  A_360_01_SQ4_A428_7_VOL : FbAnalogInput_Medium (2094) := (                _sDescription := 'Faktisk luftmengde',                 _rCov_Increment := 1,                 _eUnits := WagoTypesBacnet.eBACnetUnits.UNIT_CUBIC_METERS_PER_HOUR           );
  A_360_01_SQ4_A428_7_SP : FbAnalogValue_Medium (2141) := (                _sDescription := 'Settpunkt',                 _rCov_Increment := 1,                 _eUnits := WagoTypesBacnet.eBACnetUnits.UNIT_CUBIC_METERS_PER_HOUR           );
  A_360_01_SQ4_A428_7_VMIN : FbAnalogValue_Medium (2142) := (                _sDescription := 'Minste luftmengde',                 _rCov_Increment := 1,                 _eUnits := WagoTypesBacnet.eBACnetUnits.UNIT_CUBIC_METERS_PER_HOUR           );
  A_360_01_SQ4_A428_7_VMAX : FbAnalogValue_Medium (2143) := (                _sDescription := 'Største luftmengde',                 _rCov_Increment := 1,                 _eUnits := WagoTypesBacnet.eBACnetUnits.UNIT_CUBIC_METERS_PER_HOUR           );
  A_360_01_SQ4_A428_7_FB : FbAnalogInput_Medium (2095) := (                _sDescription := 'Spjeldvinkel',                 _rCov_Increment := 1,                 _eUnits := WagoTypesBacnet.eBACnetUnits.UNIT_PERCENT           );
  A_360_01_SQ4_A428_7_C : FbAnalogOutput_Medium (2047) := (                _sDescription := 'Pådrag',                 _rCov_Increment := 1,                 _eUnits := WagoTypesBacnet.eBACnetUnits.UNIT_PERCENT           );
  A_360_01_SQ4_A428_7_KMD : FbMultiStateValue_Large (2047) := (                _sDescription := 'Manuell overstyring',                 _udiNumberOfStates := 8           );
  A_360_01_SQ4_A428_7_OPT_EKSKL : FbBinaryValue_Medium (2047) := (                _sDescription := 'Optimizer',                 _sActiveText := 'Utkoblet',                 _sInactiveText := 'Innkoblet'           );
  A_360_01_SQ4_A428_7_A1 : FbBinaryInput_Large (2094) := (                _sDescription := 'Luftmengde Sjeld',                 _sActiveText := 'Feil på luftmengde',                 _sInactiveText := 'Ingen feil',                 _udiNotificationClass := 22           );
  A_360_01_SQ4_A428_7_A2 : FbBinaryInput_Large (2095) := (                _sDescription := 'Kommunikasjonovervåking',                 _sActiveText := 'Kommunikasjonsfeil',                 _sInactiveText := 'Ingen feil',                 _udiNotificationClass := 22           );
  B_360_02_SQ5_UBH1_VOL : FbAnalogInput_Medium (2096) := (                _sDescription := 'Faktisk luftmengde',                 _rCov_Increment := 1,                 _eUnits := WagoTypesBacnet.eBACnetUnits.UNIT_CUBIC_METERS_PER_HOUR           );
  B_360_02_SQ5_UBH1_SP : FbAnalogValue_Medium (2144) := (                _sDescription := 'Settpunkt',                 _rCov_Increment := 1,                 _eUnits := WagoTypesBacnet.eBACnetUnits.UNIT_CUBIC_METERS_PER_HOUR           );
  B_360_02_SQ5_UBH1_VMIN : FbAnalogValue_Medium (2145) := (                _sDescription := 'Minste luftmengde',                 _rCov_Increment := 1,                 _eUnits := WagoTypesBacnet.eBACnetUnits.UNIT_CUBIC_METERS_PER_HOUR           );
  B_360_02_SQ5_UBH1_VMAX : FbAnalogValue_Medium (2146) := (                _sDescription := 'Største luftmengde',                 _rCov_Increment := 1,                 _eUnits := WagoTypesBacnet.eBACnetUnits.UNIT_CUBIC_METERS_PER_HOUR           );
  B_360_02_SQ5_UBH1_FB : FbAnalogInput_Medium (2097) := (                _sDescription := 'Spjeldvinkel',                 _rCov_Increment := 1,                 _eUnits := WagoTypesBacnet.eBACnetUnits.UNIT_PERCENT           );
  B_360_02_SQ5_UBH1_C : FbAnalogOutput_Medium (2048) := (                _sDescription := 'Pådrag',                 _rCov_Increment := 1,                 _eUnits := WagoTypesBacnet.eBACnetUnits.UNIT_PERCENT           );
  B_360_02_SQ5_UBH1_KMD : FbMultiStateValue_Large (2048) := (                _sDescription := 'Manuell overstyring',                 _udiNumberOfStates := 8           );
  B_360_02_SQ5_UBH1_OPT_EKSKL : FbBinaryValue_Medium (2048) := (                _sDescription := 'Optimizer',                 _sActiveText := 'Utkoblet',                 _sInactiveText := 'Innkoblet'           );
  B_360_02_SQ5_UBH1_A1 : FbBinaryInput_Large (2096) := (                _sDescription := 'Luftmengde Sjeld',                 _sActiveText := 'Feil på luftmengde',                 _sInactiveText := 'Ingen feil',                 _udiNotificationClass := 22           );
  B_360_02_SQ5_UBH1_A2 : FbBinaryInput_Large (2097) := (                _sDescription := 'Kommunikasjonovervåking',                 _sActiveText := 'Kommunikasjonsfeil',                 _sInactiveText := 'Ingen feil',                 _udiNotificationClass := 22           );
  B_360_02_SQ5_UBH2_VOL : FbAnalogInput_Medium (2098) := (                _sDescription := 'Faktisk luftmengde',                 _rCov_Increment := 1,                 _eUnits := WagoTypesBacnet.eBACnetUnits.UNIT_CUBIC_METERS_PER_HOUR           );
  B_360_02_SQ5_UBH2_SP : FbAnalogValue_Medium (2147) := (                _sDescription := 'Settpunkt',                 _rCov_Increment := 1,                 _eUnits := WagoTypesBacnet.eBACnetUnits.UNIT_CUBIC_METERS_PER_HOUR           );
  B_360_02_SQ5_UBH2_VMIN : FbAnalogValue_Medium (2148) := (                _sDescription := 'Minste luftmengde',                 _rCov_Increment := 1,                 _eUnits := WagoTypesBacnet.eBACnetUnits.UNIT_CUBIC_METERS_PER_HOUR           );
  B_360_02_SQ5_UBH2_VMAX : FbAnalogValue_Medium (2149) := (                _sDescription := 'Største luftmengde',                 _rCov_Increment := 1,                 _eUnits := WagoTypesBacnet.eBACnetUnits.UNIT_CUBIC_METERS_PER_HOUR           );
  B_360_02_SQ5_UBH2_FB : FbAnalogInput_Medium (2099) := (                _sDescription := 'Spjeldvinkel',                 _rCov_Increment := 1,                 _eUnits := WagoTypesBacnet.eBACnetUnits.UNIT_PERCENT           );
  B_360_02_SQ5_UBH2_C : FbAnalogOutput_Medium (2049) := (                _sDescription := 'Pådrag',                 _rCov_Increment := 1,                 _eUnits := WagoTypesBacnet.eBACnetUnits.UNIT_PERCENT           );
  B_360_02_SQ5_UBH2_KMD : FbMultiStateValue_Large (2049) := (                _sDescription := 'Manuell overstyring',                 _udiNumberOfStates := 8           );
  B_360_02_SQ5_UBH2_OPT_EKSKL : FbBinaryValue_Medium (2049) := (                _sDescription := 'Optimizer',                 _sActiveText := 'Utkoblet',                 _sInactiveText := 'Innkoblet'           );
  B_360_02_SQ5_UBH2_A1 : FbBinaryInput_Large (2098) := (                _sDescription := 'Luftmengde Sjeld',                 _sActiveText := 'Feil på luftmengde',                 _sInactiveText := 'Ingen feil',                 _udiNotificationClass := 22           );
  B_360_02_SQ5_UBH2_A2 : FbBinaryInput_Large (2099) := (                _sDescription := 'Kommunikasjonovervåking',                 _sActiveText := 'Kommunikasjonsfeil',                 _sInactiveText := 'Ingen feil',                 _udiNotificationClass := 22           );
  B_360_02_SQ4_UBH1_VOL : FbAnalogInput_Medium (2100) := (                _sDescription := 'Faktisk luftmengde',                 _rCov_Increment := 1,                 _eUnits := WagoTypesBacnet.eBACnetUnits.UNIT_CUBIC_METERS_PER_HOUR           );
  B_360_02_SQ4_UBH1_SP : FbAnalogValue_Medium (2150) := (                _sDescription := 'Settpunkt',                 _rCov_Increment := 1,                 _eUnits := WagoTypesBacnet.eBACnetUnits.UNIT_CUBIC_METERS_PER_HOUR           );
  B_360_02_SQ4_UBH1_VMIN : FbAnalogValue_Medium (2151) := (                _sDescription := 'Minste luftmengde',                 _rCov_Increment := 1,                 _eUnits := WagoTypesBacnet.eBACnetUnits.UNIT_CUBIC_METERS_PER_HOUR           );
  B_360_02_SQ4_UBH1_VMAX : FbAnalogValue_Medium (2152) := (                _sDescription := 'Største luftmengde',                 _rCov_Increment := 1,                 _eUnits := WagoTypesBacnet.eBACnetUnits.UNIT_CUBIC_METERS_PER_HOUR           );
  B_360_02_SQ4_UBH1_FB : FbAnalogInput_Medium (2101) := (                _sDescription := 'Spjeldvinkel',                 _rCov_Increment := 1,                 _eUnits := WagoTypesBacnet.eBACnetUnits.UNIT_PERCENT           );
  B_360_02_SQ4_UBH1_C : FbAnalogOutput_Medium (2050) := (                _sDescription := 'Pådrag',                 _rCov_Increment := 1,                 _eUnits := WagoTypesBacnet.eBACnetUnits.UNIT_PERCENT           );
  B_360_02_SQ4_UBH1_KMD : FbMultiStateValue_Large (2050) := (                _sDescription := 'Manuell overstyring',                 _udiNumberOfStates := 8           );
  B_360_02_SQ4_UBH1_OPT_EKSKL : FbBinaryValue_Medium (2050) := (                _sDescription := 'Optimizer',                 _sActiveText := 'Utkoblet',                 _sInactiveText := 'Innkoblet'           );
  B_360_02_SQ4_UBH1_A1 : FbBinaryInput_Large (2100) := (                _sDescription := 'Luftmengde Sjeld',                 _sActiveText := 'Feil på luftmengde',                 _sInactiveText := 'Ingen feil',                 _udiNotificationClass := 22           );
  B_360_02_SQ4_UBH1_A2 : FbBinaryInput_Large (2101) := (                _sDescription := 'Kommunikasjonovervåking',                 _sActiveText := 'Kommunikasjonsfeil',                 _sInactiveText := 'Ingen feil',                 _udiNotificationClass := 22           );
  B_360_02_SQ4_UBH2_VOL : FbAnalogInput_Medium (2102) := (                _sDescription := 'Faktisk luftmengde',                 _rCov_Increment := 1,                 _eUnits := WagoTypesBacnet.eBACnetUnits.UNIT_CUBIC_METERS_PER_HOUR           );
  B_360_02_SQ4_UBH2_SP : FbAnalogValue_Medium (2153) := (                _sDescription := 'Settpunkt',                 _rCov_Increment := 1,                 _eUnits := WagoTypesBacnet.eBACnetUnits.UNIT_CUBIC_METERS_PER_HOUR           );
  B_360_02_SQ4_UBH2_VMIN : FbAnalogValue_Medium (2154) := (                _sDescription := 'Minste luftmengde',                 _rCov_Increment := 1,                 _eUnits := WagoTypesBacnet.eBACnetUnits.UNIT_CUBIC_METERS_PER_HOUR           );
  B_360_02_SQ4_UBH2_VMAX : FbAnalogValue_Medium (2155) := (                _sDescription := 'Største luftmengde',                 _rCov_Increment := 1,                 _eUnits := WagoTypesBacnet.eBACnetUnits.UNIT_CUBIC_METERS_PER_HOUR           );
  B_360_02_SQ4_UBH2_FB : FbAnalogInput_Medium (2103) := (                _sDescription := 'Spjeldvinkel',                 _rCov_Increment := 1,                 _eUnits := WagoTypesBacnet.eBACnetUnits.UNIT_PERCENT           );
  B_360_02_SQ4_UBH2_C : FbAnalogOutput_Medium (2051) := (                _sDescription := 'Pådrag',                 _rCov_Increment := 1,                 _eUnits := WagoTypesBacnet.eBACnetUnits.UNIT_PERCENT           );
  B_360_02_SQ4_UBH2_KMD : FbMultiStateValue_Large (2051) := (                _sDescription := 'Manuell overstyring',                 _udiNumberOfStates := 8           );
  B_360_02_SQ4_UBH2_OPT_EKSKL : FbBinaryValue_Medium (2051) := (                _sDescription := 'Optimizer',                 _sActiveText := 'Utkoblet',                 _sInactiveText := 'Innkoblet'           );
  B_360_02_SQ4_UBH2_A1 : FbBinaryInput_Large (2102) := (                _sDescription := 'Luftmengde Sjeld',                 _sActiveText := 'Feil på luftmengde',                 _sInactiveText := 'Ingen feil',                 _udiNotificationClass := 22           );
  B_360_02_SQ4_UBH2_A2 : FbBinaryInput_Large (2103) := (                _sDescription := 'Kommunikasjonovervåking',                 _sActiveText := 'Kommunikasjonsfeil',                 _sInactiveText := 'Ingen feil',                 _udiNotificationClass := 22           );
END_VAR

PROGRAM ClimateControl_401
  VAR
    climateController : FbMultiModeClimateControl_00_02;
    defaultSetpoints : typMultiModeClimateControllerDefaultSettings_00_01;
    dwConfigurationMask : DWORD := 2#0000_0000_0000_0000_0000_0001_0000_0010;
  END_VAR
  VAR_OUTPUT
    actualSetpointHeating : REAL;  (* Variabler kun for overvåking *)
    actualSetpointCooling : REAL;
    actualSetpointCo2 : REAL;
    meanTemp : REAL;
    meanCo2 : REAL;
    presence : BOOL;
    gainHeating : REAL;
    gainCooling : REAL;
    gainAirQuality : REAL;
    damperOutput : REAL;
    currentWorkingMode : enumMultiModeClimateActiveControlMode_00_01;
  END_VAR

                
    
// Innstillinger for rom:
IF (firstScan) THEN
    PersistentVars.typClimateControllerSettingsRoom401.ahuSystem		:= 001;
    PersistentVars.typClimateControllerSettingsRoom401.heatingSystem	:= 004;
    PersistentVars.typClimateControllerSettingsRoom401.coolingSystem	:= 004;
    defaultSetpoints 							:= PersistentVars.typClimateControlDefaultSettings;
    
// Hvis du ønsker egne innstillinger for rommet, kjør settings
    // settings();
END_IF

// Tilbakestill settpunkt (global kommando)
IF (GVL.initDefaultSettings) THEN
    climateController.setDefaultSetpoints();
END_IF

// Kjør funksjonsblokk
climateController(
    typController			:= typClimateControllerInterfaceRoom401, 
    typSettings				:= PersistentVars.typClimateControllerSettingsRoom401, 
    typDefaultSetpoints		:= defaultSetpoints,
    dwConfigurationMask		:= dwConfigurationMask            
);
        
// Registrer temperaturer
climateController.Temp          := PRG_KnxLine_1.M1_017_401_RMA6001_TMP_ACT.rValue_OUT;
climateController.Temp          := PRG_KnxLine_1.M1_018_401_RMA6002_TMP_ACT.rValue_OUT;

// Registrer CO2
climateController.CO2          := PRG_KnxLine_1.M1_033_401_RMA6001_CO2_ACT.rValue_OUT;
climateController.CO2          := PRG_KnxLine_1.M1_034_401_RMA6002_CO2_ACT.rValue_OUT;

// Registrer tilstedeværelse
climateController.Presence          := PRG_KnxLine_1.M1_001_401_RMA6001_MOV_ACT.xSwitch_OUT;
climateController.Presence          := PRG_KnxLine_1.M1_002_401_RMA6002_MOV_ACT.xSwitch_OUT;

meanTemp					:= typClimateControllerInterfaceRoom401.actuators.heating.processValue;
meanCo2						:= climateController.Co2;
presence					:= climateController.Presence;

actualSetpointHeating 		:= typClimateControllerInterfaceRoom401.actuators.heating.setpoint;
gainHeating 				:= typClimateControllerInterfaceRoom401.actuators.heating.controlledVariable;

actualSetpointCooling 		:= typClimateControllerInterfaceRoom401.actuators.cooling.setpoint;
gainCooling 				:= typClimateControllerInterfaceRoom401.actuators.cooling.controlledVariable;

actualSetpointCo2			:= typClimateControllerInterfaceRoom401.actuators.airQuality.setpoint;
gainAirQuality				:= typClimateControllerInterfaceRoom401.actuators.airQuality.controlledVariable; 
damperOutput				:= typClimateControllerInterfaceRoom401.actuators.damper.setpoint;

currentWorkingMode			:= typClimateControllerInterfaceRoom401.currentMode;                   
                
                
              

ACTION settings:
                            
                                
defaultSetpoints.heating.comfort.setpoint	:= 21;
defaultSetpoints.heating.standby.setpoint	:= 2;
defaultSetpoints.heating.economy.setpoint	:= 3;
defaultSetpoints.cooling.comfort.setpoint	:= 2;
defaultSetpoints.cooling.standby.setpoint	:= 3;
defaultSetpoints.cooling.economy.setpoint	:= 4;
defaultSetpoints.co2.comfort.setpoint		:= 600;
defaultSetpoints.presenceDelayOff			:= 30;
defaultSetpoints.heating.pidSettings.KP		:= 1;
defaultSetpoints.heating.pidSettings.TN		:= 60;
defaultSetpoints.cooling.pidSettings.KP		:= 1;
defaultSetpoints.cooling.pidSettings.TN		:= 60;
defaultSetpoints.co2.pidSettings.KP			:= 20;
defaultSetpoints.co2.pidSettings.TN			:= 4000;
                            
                        
END_ACTION
END_PROGRAM

PROGRAM ClimateControl_406
  VAR
    climateController : FbMultiModeClimateControl_00_02;
    defaultSetpoints : typMultiModeClimateControllerDefaultSettings_00_01;
    dwConfigurationMask : DWORD := 2#0000_0000_0000_0000_0000_0001_0000_0010;
  END_VAR
  VAR_OUTPUT
    actualSetpointHeating : REAL;  (* Variabler kun for overvåking *)
    actualSetpointCooling : REAL;
    actualSetpointCo2 : REAL;
    meanTemp : REAL;
    meanCo2 : REAL;
    presence : BOOL;
    gainHeating : REAL;
    gainCooling : REAL;
    gainAirQuality : REAL;
    damperOutput : REAL;
    currentWorkingMode : enumMultiModeClimateActiveControlMode_00_01;
  END_VAR

                
    
// Innstillinger for rom:
IF (firstScan) THEN
    PersistentVars.typClimateControllerSettingsRoom406.ahuSystem		:= 001;
    PersistentVars.typClimateControllerSettingsRoom406.heatingSystem	:= 004;
    PersistentVars.typClimateControllerSettingsRoom406.coolingSystem	:= 004;
    defaultSetpoints 							:= PersistentVars.typClimateControlDefaultSettings;
    
// Hvis du ønsker egne innstillinger for rommet, kjør settings
    // settings();
END_IF

// Tilbakestill settpunkt (global kommando)
IF (GVL.initDefaultSettings) THEN
    climateController.setDefaultSetpoints();
END_IF

// Kjør funksjonsblokk
climateController(
    typController			:= typClimateControllerInterfaceRoom406, 
    typSettings				:= PersistentVars.typClimateControllerSettingsRoom406, 
    typDefaultSetpoints		:= defaultSetpoints,
    dwConfigurationMask		:= dwConfigurationMask            
);
        
// Registrer temperaturer
climateController.Temp          := PRG_KnxLine_1.M1_019_406_RMA6003_TMP_ACT.rValue_OUT;

// Registrer CO2
climateController.CO2          := PRG_KnxLine_1.M1_035_406_RMA6003_CO2_ACT.rValue_OUT;

// Registrer tilstedeværelse
climateController.Presence          := PRG_KnxLine_1.M1_003_406_RMA6003_MOV_ACT.xSwitch_OUT;

meanTemp					:= typClimateControllerInterfaceRoom406.actuators.heating.processValue;
meanCo2						:= climateController.Co2;
presence					:= climateController.Presence;

actualSetpointHeating 		:= typClimateControllerInterfaceRoom406.actuators.heating.setpoint;
gainHeating 				:= typClimateControllerInterfaceRoom406.actuators.heating.controlledVariable;

actualSetpointCooling 		:= typClimateControllerInterfaceRoom406.actuators.cooling.setpoint;
gainCooling 				:= typClimateControllerInterfaceRoom406.actuators.cooling.controlledVariable;

actualSetpointCo2			:= typClimateControllerInterfaceRoom406.actuators.airQuality.setpoint;
gainAirQuality				:= typClimateControllerInterfaceRoom406.actuators.airQuality.controlledVariable; 
damperOutput				:= typClimateControllerInterfaceRoom406.actuators.damper.setpoint;

currentWorkingMode			:= typClimateControllerInterfaceRoom406.currentMode;                   
                
                
              

ACTION settings:
                            
                                
defaultSetpoints.heating.comfort.setpoint	:= 21;
defaultSetpoints.heating.standby.setpoint	:= 2;
defaultSetpoints.heating.economy.setpoint	:= 3;
defaultSetpoints.cooling.comfort.setpoint	:= 2;
defaultSetpoints.cooling.standby.setpoint	:= 3;
defaultSetpoints.cooling.economy.setpoint	:= 4;
defaultSetpoints.co2.comfort.setpoint		:= 600;
defaultSetpoints.presenceDelayOff			:= 30;
defaultSetpoints.heating.pidSettings.KP		:= 1;
defaultSetpoints.heating.pidSettings.TN		:= 60;
defaultSetpoints.cooling.pidSettings.KP		:= 1;
defaultSetpoints.cooling.pidSettings.TN		:= 60;
defaultSetpoints.co2.pidSettings.KP			:= 20;
defaultSetpoints.co2.pidSettings.TN			:= 4000;
                            
                        
END_ACTION
END_PROGRAM

PROGRAM ClimateControl_407
  VAR
    climateController : FbMultiModeClimateControl_00_02;
    defaultSetpoints : typMultiModeClimateControllerDefaultSettings_00_01;
    dwConfigurationMask : DWORD := 2#0000_0000_0000_0000_0000_0001_0000_0010;
  END_VAR
  VAR_OUTPUT
    actualSetpointHeating : REAL;  (* Variabler kun for overvåking *)
    actualSetpointCooling : REAL;
    actualSetpointCo2 : REAL;
    meanTemp : REAL;
    meanCo2 : REAL;
    presence : BOOL;
    gainHeating : REAL;
    gainCooling : REAL;
    gainAirQuality : REAL;
    damperOutput : REAL;
    currentWorkingMode : enumMultiModeClimateActiveControlMode_00_01;
  END_VAR

                
    
// Innstillinger for rom:
IF (firstScan) THEN
    PersistentVars.typClimateControllerSettingsRoom407.ahuSystem		:= 001;
    PersistentVars.typClimateControllerSettingsRoom407.heatingSystem	:= 004;
    PersistentVars.typClimateControllerSettingsRoom407.coolingSystem	:= 004;
    defaultSetpoints 							:= PersistentVars.typClimateControlDefaultSettings;
    
// Hvis du ønsker egne innstillinger for rommet, kjør settings
    // settings();
END_IF

// Tilbakestill settpunkt (global kommando)
IF (GVL.initDefaultSettings) THEN
    climateController.setDefaultSetpoints();
END_IF

// Kjør funksjonsblokk
climateController(
    typController			:= typClimateControllerInterfaceRoom407, 
    typSettings				:= PersistentVars.typClimateControllerSettingsRoom407, 
    typDefaultSetpoints		:= defaultSetpoints,
    dwConfigurationMask		:= dwConfigurationMask            
);
        
// Registrer temperaturer
climateController.Temp          := PRG_KnxLine_1.M1_020_407_RMA6004_TMP_ACT.rValue_OUT;

// Registrer CO2
climateController.CO2          := PRG_KnxLine_1.M1_036_407_RMA6004_CO2_ACT.rValue_OUT;

// Registrer tilstedeværelse
climateController.Presence          := PRG_KnxLine_1.M1_004_407_RMA6004_MOV_ACT.xSwitch_OUT;

meanTemp					:= typClimateControllerInterfaceRoom407.actuators.heating.processValue;
meanCo2						:= climateController.Co2;
presence					:= climateController.Presence;

actualSetpointHeating 		:= typClimateControllerInterfaceRoom407.actuators.heating.setpoint;
gainHeating 				:= typClimateControllerInterfaceRoom407.actuators.heating.controlledVariable;

actualSetpointCooling 		:= typClimateControllerInterfaceRoom407.actuators.cooling.setpoint;
gainCooling 				:= typClimateControllerInterfaceRoom407.actuators.cooling.controlledVariable;

actualSetpointCo2			:= typClimateControllerInterfaceRoom407.actuators.airQuality.setpoint;
gainAirQuality				:= typClimateControllerInterfaceRoom407.actuators.airQuality.controlledVariable; 
damperOutput				:= typClimateControllerInterfaceRoom407.actuators.damper.setpoint;

currentWorkingMode			:= typClimateControllerInterfaceRoom407.currentMode;                   
                
                
              

ACTION settings:
                            
                                
defaultSetpoints.heating.comfort.setpoint	:= 21;
defaultSetpoints.heating.standby.setpoint	:= 2;
defaultSetpoints.heating.economy.setpoint	:= 3;
defaultSetpoints.cooling.comfort.setpoint	:= 2;
defaultSetpoints.cooling.standby.setpoint	:= 3;
defaultSetpoints.cooling.economy.setpoint	:= 4;
defaultSetpoints.co2.comfort.setpoint		:= 600;
defaultSetpoints.presenceDelayOff			:= 30;
defaultSetpoints.heating.pidSettings.KP		:= 1;
defaultSetpoints.heating.pidSettings.TN		:= 60;
defaultSetpoints.cooling.pidSettings.KP		:= 1;
defaultSetpoints.cooling.pidSettings.TN		:= 60;
defaultSetpoints.co2.pidSettings.KP			:= 20;
defaultSetpoints.co2.pidSettings.TN			:= 4000;
                            
                        
END_ACTION
END_PROGRAM

PROGRAM ClimateControl_408
  VAR
    climateController : FbMultiModeClimateControl_00_02;
    defaultSetpoints : typMultiModeClimateControllerDefaultSettings_00_01;
    dwConfigurationMask : DWORD := 2#0000_0000_0000_0000_0000_0001_0000_0010;
  END_VAR
  VAR_OUTPUT
    actualSetpointHeating : REAL;  (* Variabler kun for overvåking *)
    actualSetpointCooling : REAL;
    actualSetpointCo2 : REAL;
    meanTemp : REAL;
    meanCo2 : REAL;
    presence : BOOL;
    gainHeating : REAL;
    gainCooling : REAL;
    gainAirQuality : REAL;
    damperOutput : REAL;
    currentWorkingMode : enumMultiModeClimateActiveControlMode_00_01;
  END_VAR

                
    
// Innstillinger for rom:
IF (firstScan) THEN
    PersistentVars.typClimateControllerSettingsRoom408.ahuSystem		:= 001;
    PersistentVars.typClimateControllerSettingsRoom408.heatingSystem	:= 004;
    PersistentVars.typClimateControllerSettingsRoom408.coolingSystem	:= 004;
    defaultSetpoints 							:= PersistentVars.typClimateControlDefaultSettings;
    
// Hvis du ønsker egne innstillinger for rommet, kjør settings
    // settings();
END_IF

// Tilbakestill settpunkt (global kommando)
IF (GVL.initDefaultSettings) THEN
    climateController.setDefaultSetpoints();
END_IF

// Kjør funksjonsblokk
climateController(
    typController			:= typClimateControllerInterfaceRoom408, 
    typSettings				:= PersistentVars.typClimateControllerSettingsRoom408, 
    typDefaultSetpoints		:= defaultSetpoints,
    dwConfigurationMask		:= dwConfigurationMask            
);
        
// Registrer temperaturer
climateController.Temp          := PRG_KnxLine_1.M1_021_408_RMA6005_TMP_ACT.rValue_OUT;

// Registrer CO2
climateController.CO2          := PRG_KnxLine_1.M1_037_408_RMA6005_CO2_ACT.rValue_OUT;

// Registrer tilstedeværelse
climateController.Presence          := PRG_KnxLine_1.M1_005_408_RMA6005_MOV_ACT.xSwitch_OUT;

meanTemp					:= typClimateControllerInterfaceRoom408.actuators.heating.processValue;
meanCo2						:= climateController.Co2;
presence					:= climateController.Presence;

actualSetpointHeating 		:= typClimateControllerInterfaceRoom408.actuators.heating.setpoint;
gainHeating 				:= typClimateControllerInterfaceRoom408.actuators.heating.controlledVariable;

actualSetpointCooling 		:= typClimateControllerInterfaceRoom408.actuators.cooling.setpoint;
gainCooling 				:= typClimateControllerInterfaceRoom408.actuators.cooling.controlledVariable;

actualSetpointCo2			:= typClimateControllerInterfaceRoom408.actuators.airQuality.setpoint;
gainAirQuality				:= typClimateControllerInterfaceRoom408.actuators.airQuality.controlledVariable; 
damperOutput				:= typClimateControllerInterfaceRoom408.actuators.damper.setpoint;

currentWorkingMode			:= typClimateControllerInterfaceRoom408.currentMode;                   
                
                
              

ACTION settings:
                            
                                
defaultSetpoints.heating.comfort.setpoint	:= 21;
defaultSetpoints.heating.standby.setpoint	:= 2;
defaultSetpoints.heating.economy.setpoint	:= 3;
defaultSetpoints.cooling.comfort.setpoint	:= 2;
defaultSetpoints.cooling.standby.setpoint	:= 3;
defaultSetpoints.cooling.economy.setpoint	:= 4;
defaultSetpoints.co2.comfort.setpoint		:= 600;
defaultSetpoints.presenceDelayOff			:= 30;
defaultSetpoints.heating.pidSettings.KP		:= 1;
defaultSetpoints.heating.pidSettings.TN		:= 60;
defaultSetpoints.cooling.pidSettings.KP		:= 1;
defaultSetpoints.cooling.pidSettings.TN		:= 60;
defaultSetpoints.co2.pidSettings.KP			:= 20;
defaultSetpoints.co2.pidSettings.TN			:= 4000;
                            
                        
END_ACTION
END_PROGRAM

PROGRAM ClimateControl_409
  VAR
    climateController : FbMultiModeClimateControl_00_02;
    defaultSetpoints : typMultiModeClimateControllerDefaultSettings_00_01;
    dwConfigurationMask : DWORD := 2#0000_0000_0000_0000_0000_0001_0000_0010;
  END_VAR
  VAR_OUTPUT
    actualSetpointHeating : REAL;  (* Variabler kun for overvåking *)
    actualSetpointCooling : REAL;
    actualSetpointCo2 : REAL;
    meanTemp : REAL;
    meanCo2 : REAL;
    presence : BOOL;
    gainHeating : REAL;
    gainCooling : REAL;
    gainAirQuality : REAL;
    damperOutput : REAL;
    currentWorkingMode : enumMultiModeClimateActiveControlMode_00_01;
  END_VAR

                
    
// Innstillinger for rom:
IF (firstScan) THEN
    PersistentVars.typClimateControllerSettingsRoom409.ahuSystem		:= 001;
    PersistentVars.typClimateControllerSettingsRoom409.heatingSystem	:= 004;
    PersistentVars.typClimateControllerSettingsRoom409.coolingSystem	:= 004;
    defaultSetpoints 							:= PersistentVars.typClimateControlDefaultSettings;
    
// Hvis du ønsker egne innstillinger for rommet, kjør settings
    // settings();
END_IF

// Tilbakestill settpunkt (global kommando)
IF (GVL.initDefaultSettings) THEN
    climateController.setDefaultSetpoints();
END_IF

// Kjør funksjonsblokk
climateController(
    typController			:= typClimateControllerInterfaceRoom409, 
    typSettings				:= PersistentVars.typClimateControllerSettingsRoom409, 
    typDefaultSetpoints		:= defaultSetpoints,
    dwConfigurationMask		:= dwConfigurationMask            
);
        
// Registrer temperaturer
climateController.Temp          := PRG_KnxLine_1.M1_022_409_RMA6006_TMP_ACT.rValue_OUT;
climateController.Temp          := PRG_KnxLine_1.M1_023_409_RMA6007_TMP_ACT.rValue_OUT;
climateController.Temp          := PRG_KnxLine_1.M1_024_409_RMA6008_TMP_ACT.rValue_OUT;

// Registrer CO2
climateController.CO2          := PRG_KnxLine_1.M1_038_409_RMA6006_CO2_ACT.rValue_OUT;
climateController.CO2          := PRG_KnxLine_1.M1_039_409_RMA6007_CO2_ACT.rValue_OUT;
climateController.CO2          := PRG_KnxLine_1.M1_040_409_RMA6008_CO2_ACT.rValue_OUT;

// Registrer tilstedeværelse
climateController.Presence          := PRG_KnxLine_1.M1_006_409_RMA6006_MOV_ACT.xSwitch_OUT;
climateController.Presence          := PRG_KnxLine_1.M1_007_409_RMA6007_MOV_ACT.xSwitch_OUT;
climateController.Presence          := PRG_KnxLine_1.M1_008_409_RMA6008_MOV_ACT.xSwitch_OUT;

meanTemp					:= typClimateControllerInterfaceRoom409.actuators.heating.processValue;
meanCo2						:= climateController.Co2;
presence					:= climateController.Presence;

actualSetpointHeating 		:= typClimateControllerInterfaceRoom409.actuators.heating.setpoint;
gainHeating 				:= typClimateControllerInterfaceRoom409.actuators.heating.controlledVariable;

actualSetpointCooling 		:= typClimateControllerInterfaceRoom409.actuators.cooling.setpoint;
gainCooling 				:= typClimateControllerInterfaceRoom409.actuators.cooling.controlledVariable;

actualSetpointCo2			:= typClimateControllerInterfaceRoom409.actuators.airQuality.setpoint;
gainAirQuality				:= typClimateControllerInterfaceRoom409.actuators.airQuality.controlledVariable; 
damperOutput				:= typClimateControllerInterfaceRoom409.actuators.damper.setpoint;

currentWorkingMode			:= typClimateControllerInterfaceRoom409.currentMode;                   
                
                
              

ACTION settings:
                            
                                
defaultSetpoints.heating.comfort.setpoint	:= 21;
defaultSetpoints.heating.standby.setpoint	:= 2;
defaultSetpoints.heating.economy.setpoint	:= 3;
defaultSetpoints.cooling.comfort.setpoint	:= 2;
defaultSetpoints.cooling.standby.setpoint	:= 3;
defaultSetpoints.cooling.economy.setpoint	:= 4;
defaultSetpoints.co2.comfort.setpoint		:= 600;
defaultSetpoints.presenceDelayOff			:= 30;
defaultSetpoints.heating.pidSettings.KP		:= 1;
defaultSetpoints.heating.pidSettings.TN		:= 60;
defaultSetpoints.cooling.pidSettings.KP		:= 1;
defaultSetpoints.cooling.pidSettings.TN		:= 60;
defaultSetpoints.co2.pidSettings.KP			:= 20;
defaultSetpoints.co2.pidSettings.TN			:= 4000;
                            
                        
END_ACTION
END_PROGRAM

PROGRAM ClimateControl_464
  VAR
    climateController : FbMultiModeClimateControl_00_02;
    defaultSetpoints : typMultiModeClimateControllerDefaultSettings_00_01;
    dwConfigurationMask : DWORD := 2#0000_0000_0000_0000_0000_0001_0000_0010;
  END_VAR
  VAR_OUTPUT
    actualSetpointHeating : REAL;  (* Variabler kun for overvåking *)
    actualSetpointCooling : REAL;
    actualSetpointCo2 : REAL;
    meanTemp : REAL;
    meanCo2 : REAL;
    presence : BOOL;
    gainHeating : REAL;
    gainCooling : REAL;
    gainAirQuality : REAL;
    damperOutput : REAL;
    currentWorkingMode : enumMultiModeClimateActiveControlMode_00_01;
  END_VAR

                
    
// Innstillinger for rom:
IF (firstScan) THEN
    PersistentVars.typClimateControllerSettingsRoom464.ahuSystem		:= 001;
    PersistentVars.typClimateControllerSettingsRoom464.heatingSystem	:= 004;
    PersistentVars.typClimateControllerSettingsRoom464.coolingSystem	:= 004;
    defaultSetpoints 							:= PersistentVars.typClimateControlDefaultSettings;
    
// Hvis du ønsker egne innstillinger for rommet, kjør settings
    // settings();
END_IF

// Tilbakestill settpunkt (global kommando)
IF (GVL.initDefaultSettings) THEN
    climateController.setDefaultSetpoints();
END_IF

// Kjør funksjonsblokk
climateController(
    typController			:= typClimateControllerInterfaceRoom464, 
    typSettings				:= PersistentVars.typClimateControllerSettingsRoom464, 
    typDefaultSetpoints		:= defaultSetpoints,
    dwConfigurationMask		:= dwConfigurationMask            
);
        
// Registrer temperaturer
climateController.Temp          := PRG_KnxLine_1.M1_025_464_RMA6009_TMP_ACT.rValue_OUT;
climateController.Temp          := PRG_KnxLine_1.M1_026_464_RMA6010_TMP_ACT.rValue_OUT;

// Registrer CO2
climateController.CO2          := PRG_KnxLine_1.M1_041_464_RMA6009_CO2_ACT.rValue_OUT;
climateController.CO2          := PRG_KnxLine_1.M1_042_464_RMA6010_CO2_ACT.rValue_OUT;

// Registrer tilstedeværelse
climateController.Presence          := PRG_KnxLine_1.M1_009_464_RMA6009_MOV_ACT.xSwitch_OUT;
climateController.Presence          := PRG_KnxLine_1.M1_010_464_RMA6010_MOV_ACT.xSwitch_OUT;

meanTemp					:= typClimateControllerInterfaceRoom464.actuators.heating.processValue;
meanCo2						:= climateController.Co2;
presence					:= climateController.Presence;

actualSetpointHeating 		:= typClimateControllerInterfaceRoom464.actuators.heating.setpoint;
gainHeating 				:= typClimateControllerInterfaceRoom464.actuators.heating.controlledVariable;

actualSetpointCooling 		:= typClimateControllerInterfaceRoom464.actuators.cooling.setpoint;
gainCooling 				:= typClimateControllerInterfaceRoom464.actuators.cooling.controlledVariable;

actualSetpointCo2			:= typClimateControllerInterfaceRoom464.actuators.airQuality.setpoint;
gainAirQuality				:= typClimateControllerInterfaceRoom464.actuators.airQuality.controlledVariable; 
damperOutput				:= typClimateControllerInterfaceRoom464.actuators.damper.setpoint;

currentWorkingMode			:= typClimateControllerInterfaceRoom464.currentMode;                   
                
                
              

ACTION settings:
                            
                                
defaultSetpoints.heating.comfort.setpoint	:= 21;
defaultSetpoints.heating.standby.setpoint	:= 2;
defaultSetpoints.heating.economy.setpoint	:= 3;
defaultSetpoints.cooling.comfort.setpoint	:= 2;
defaultSetpoints.cooling.standby.setpoint	:= 3;
defaultSetpoints.cooling.economy.setpoint	:= 4;
defaultSetpoints.co2.comfort.setpoint		:= 600;
defaultSetpoints.presenceDelayOff			:= 30;
defaultSetpoints.heating.pidSettings.KP		:= 1;
defaultSetpoints.heating.pidSettings.TN		:= 60;
defaultSetpoints.cooling.pidSettings.KP		:= 1;
defaultSetpoints.cooling.pidSettings.TN		:= 60;
defaultSetpoints.co2.pidSettings.KP			:= 20;
defaultSetpoints.co2.pidSettings.TN			:= 4000;
                            
                        
END_ACTION
END_PROGRAM

PROGRAM ClimateControl_415
  VAR
    climateController : FbMultiModeClimateControl_00_02;
    defaultSetpoints : typMultiModeClimateControllerDefaultSettings_00_01;
    dwConfigurationMask : DWORD := 2#0000_0000_0000_0000_0000_0001_0000_0010;
  END_VAR
  VAR_OUTPUT
    actualSetpointHeating : REAL;  (* Variabler kun for overvåking *)
    actualSetpointCooling : REAL;
    actualSetpointCo2 : REAL;
    meanTemp : REAL;
    meanCo2 : REAL;
    presence : BOOL;
    gainHeating : REAL;
    gainCooling : REAL;
    gainAirQuality : REAL;
    damperOutput : REAL;
    currentWorkingMode : enumMultiModeClimateActiveControlMode_00_01;
  END_VAR

                
    
// Innstillinger for rom:
IF (firstScan) THEN
    PersistentVars.typClimateControllerSettingsRoom415.ahuSystem		:= 001;
    PersistentVars.typClimateControllerSettingsRoom415.heatingSystem	:= 004;
    PersistentVars.typClimateControllerSettingsRoom415.coolingSystem	:= 004;
    defaultSetpoints 							:= PersistentVars.typClimateControlDefaultSettings;
    
// Hvis du ønsker egne innstillinger for rommet, kjør settings
    // settings();
END_IF

// Tilbakestill settpunkt (global kommando)
IF (GVL.initDefaultSettings) THEN
    climateController.setDefaultSetpoints();
END_IF

// Kjør funksjonsblokk
climateController(
    typController			:= typClimateControllerInterfaceRoom415, 
    typSettings				:= PersistentVars.typClimateControllerSettingsRoom415, 
    typDefaultSetpoints		:= defaultSetpoints,
    dwConfigurationMask		:= dwConfigurationMask            
);
        
// Registrer temperaturer
climateController.Temp          := PRG_KnxLine_1.M1_027_415_RMA6011_TMP_ACT.rValue_OUT;

// Registrer CO2
climateController.CO2          := PRG_KnxLine_1.M1_043_415_RMA6011_CO2_ACT.rValue_OUT;

// Registrer tilstedeværelse
climateController.Presence          := PRG_KnxLine_1.M1_011_415_RMA6011_MOV_ACT.xSwitch_OUT;

meanTemp					:= typClimateControllerInterfaceRoom415.actuators.heating.processValue;
meanCo2						:= climateController.Co2;
presence					:= climateController.Presence;

actualSetpointHeating 		:= typClimateControllerInterfaceRoom415.actuators.heating.setpoint;
gainHeating 				:= typClimateControllerInterfaceRoom415.actuators.heating.controlledVariable;

actualSetpointCooling 		:= typClimateControllerInterfaceRoom415.actuators.cooling.setpoint;
gainCooling 				:= typClimateControllerInterfaceRoom415.actuators.cooling.controlledVariable;

actualSetpointCo2			:= typClimateControllerInterfaceRoom415.actuators.airQuality.setpoint;
gainAirQuality				:= typClimateControllerInterfaceRoom415.actuators.airQuality.controlledVariable; 
damperOutput				:= typClimateControllerInterfaceRoom415.actuators.damper.setpoint;

currentWorkingMode			:= typClimateControllerInterfaceRoom415.currentMode;                   
                
                
              

ACTION settings:
                            
                                
defaultSetpoints.heating.comfort.setpoint	:= 21;
defaultSetpoints.heating.standby.setpoint	:= 2;
defaultSetpoints.heating.economy.setpoint	:= 3;
defaultSetpoints.cooling.comfort.setpoint	:= 2;
defaultSetpoints.cooling.standby.setpoint	:= 3;
defaultSetpoints.cooling.economy.setpoint	:= 4;
defaultSetpoints.co2.comfort.setpoint		:= 600;
defaultSetpoints.presenceDelayOff			:= 30;
defaultSetpoints.heating.pidSettings.KP		:= 1;
defaultSetpoints.heating.pidSettings.TN		:= 60;
defaultSetpoints.cooling.pidSettings.KP		:= 1;
defaultSetpoints.cooling.pidSettings.TN		:= 60;
defaultSetpoints.co2.pidSettings.KP			:= 20;
defaultSetpoints.co2.pidSettings.TN			:= 4000;
                            
                        
END_ACTION
END_PROGRAM

PROGRAM ClimateControl_422
  VAR
    climateController : FbMultiModeClimateControl_00_02;
    defaultSetpoints : typMultiModeClimateControllerDefaultSettings_00_01;
    dwConfigurationMask : DWORD := 2#0000_0000_0000_0000_0000_0001_0000_0010;
  END_VAR
  VAR_OUTPUT
    actualSetpointHeating : REAL;  (* Variabler kun for overvåking *)
    actualSetpointCooling : REAL;
    actualSetpointCo2 : REAL;
    meanTemp : REAL;
    meanCo2 : REAL;
    presence : BOOL;
    gainHeating : REAL;
    gainCooling : REAL;
    gainAirQuality : REAL;
    damperOutput : REAL;
    currentWorkingMode : enumMultiModeClimateActiveControlMode_00_01;
  END_VAR

                
    
// Innstillinger for rom:
IF (firstScan) THEN
    PersistentVars.typClimateControllerSettingsRoom422.ahuSystem		:= 001;
    PersistentVars.typClimateControllerSettingsRoom422.heatingSystem	:= 004;
    PersistentVars.typClimateControllerSettingsRoom422.coolingSystem	:= 004;
    defaultSetpoints 							:= PersistentVars.typClimateControlDefaultSettings;
    
// Hvis du ønsker egne innstillinger for rommet, kjør settings
    // settings();
END_IF

// Tilbakestill settpunkt (global kommando)
IF (GVL.initDefaultSettings) THEN
    climateController.setDefaultSetpoints();
END_IF

// Kjør funksjonsblokk
climateController(
    typController			:= typClimateControllerInterfaceRoom422, 
    typSettings				:= PersistentVars.typClimateControllerSettingsRoom422, 
    typDefaultSetpoints		:= defaultSetpoints,
    dwConfigurationMask		:= dwConfigurationMask            
);
        
// Registrer temperaturer
climateController.Temp          := PRG_KnxLine_1.M1_028_422_RMA6012_TMP_ACT.rValue_OUT;
climateController.Temp          := PRG_KnxLine_1.M1_029_422_RMA6013_TMP_ACT.rValue_OUT;

// Registrer CO2
climateController.CO2          := PRG_KnxLine_1.M1_044_422_RMA6012_CO2_ACT.rValue_OUT;
climateController.CO2          := PRG_KnxLine_1.M1_045_422_RMA6013_CO2_ACT.rValue_OUT;

// Registrer tilstedeværelse
climateController.Presence          := PRG_KnxLine_1.M1_012_422_RMA6012_MOV_ACT.xSwitch_OUT;
climateController.Presence          := PRG_KnxLine_1.M1_013_422_RMA6013_MOV_ACT.xSwitch_OUT;

meanTemp					:= typClimateControllerInterfaceRoom422.actuators.heating.processValue;
meanCo2						:= climateController.Co2;
presence					:= climateController.Presence;

actualSetpointHeating 		:= typClimateControllerInterfaceRoom422.actuators.heating.setpoint;
gainHeating 				:= typClimateControllerInterfaceRoom422.actuators.heating.controlledVariable;

actualSetpointCooling 		:= typClimateControllerInterfaceRoom422.actuators.cooling.setpoint;
gainCooling 				:= typClimateControllerInterfaceRoom422.actuators.cooling.controlledVariable;

actualSetpointCo2			:= typClimateControllerInterfaceRoom422.actuators.airQuality.setpoint;
gainAirQuality				:= typClimateControllerInterfaceRoom422.actuators.airQuality.controlledVariable; 
damperOutput				:= typClimateControllerInterfaceRoom422.actuators.damper.setpoint;

currentWorkingMode			:= typClimateControllerInterfaceRoom422.currentMode;                   
                
                
              

ACTION settings:
                            
                                
defaultSetpoints.heating.comfort.setpoint	:= 21;
defaultSetpoints.heating.standby.setpoint	:= 2;
defaultSetpoints.heating.economy.setpoint	:= 3;
defaultSetpoints.cooling.comfort.setpoint	:= 2;
defaultSetpoints.cooling.standby.setpoint	:= 3;
defaultSetpoints.cooling.economy.setpoint	:= 4;
defaultSetpoints.co2.comfort.setpoint		:= 600;
defaultSetpoints.presenceDelayOff			:= 30;
defaultSetpoints.heating.pidSettings.KP		:= 1;
defaultSetpoints.heating.pidSettings.TN		:= 60;
defaultSetpoints.cooling.pidSettings.KP		:= 1;
defaultSetpoints.cooling.pidSettings.TN		:= 60;
defaultSetpoints.co2.pidSettings.KP			:= 20;
defaultSetpoints.co2.pidSettings.TN			:= 4000;
                            
                        
END_ACTION
END_PROGRAM

PROGRAM ClimateControl_426_1
  VAR
    climateController : FbMultiModeClimateControl_00_02;
    defaultSetpoints : typMultiModeClimateControllerDefaultSettings_00_01;
    dwConfigurationMask : DWORD := 2#0000_0000_0000_0000_0000_0001_0000_0010;
  END_VAR
  VAR_OUTPUT
    actualSetpointHeating : REAL;  (* Variabler kun for overvåking *)
    actualSetpointCooling : REAL;
    actualSetpointCo2 : REAL;
    meanTemp : REAL;
    meanCo2 : REAL;
    presence : BOOL;
    gainHeating : REAL;
    gainCooling : REAL;
    gainAirQuality : REAL;
    damperOutput : REAL;
    currentWorkingMode : enumMultiModeClimateActiveControlMode_00_01;
  END_VAR

                
    
// Innstillinger for rom:
IF (firstScan) THEN
    PersistentVars.typClimateControllerSettingsRoom426_1.ahuSystem		:= 001;
    PersistentVars.typClimateControllerSettingsRoom426_1.heatingSystem	:= 004;
    PersistentVars.typClimateControllerSettingsRoom426_1.coolingSystem	:= 004;
    defaultSetpoints 							:= PersistentVars.typClimateControlDefaultSettings;
    
// Hvis du ønsker egne innstillinger for rommet, kjør settings
    // settings();
END_IF

// Tilbakestill settpunkt (global kommando)
IF (GVL.initDefaultSettings) THEN
    climateController.setDefaultSetpoints();
END_IF

// Kjør funksjonsblokk
climateController(
    typController			:= typClimateControllerInterfaceRoom426_1, 
    typSettings				:= PersistentVars.typClimateControllerSettingsRoom426_1, 
    typDefaultSetpoints		:= defaultSetpoints,
    dwConfigurationMask		:= dwConfigurationMask            
);
        
// Registrer temperaturer
climateController.Temp          := PRG_KnxLine_1.M1_030_426_1_RMA6014_TMP_ACT.rValue_OUT;

// Registrer CO2
climateController.CO2          := PRG_KnxLine_1.M1_046_426_1_RMA6014_CO2_ACT.rValue_OUT;

// Registrer tilstedeværelse
climateController.Presence          := PRG_KnxLine_1.M1_014_426_1_RMA6014_MOV_ACT.xSwitch_OUT;

meanTemp					:= typClimateControllerInterfaceRoom426_1.actuators.heating.processValue;
meanCo2						:= climateController.Co2;
presence					:= climateController.Presence;

actualSetpointHeating 		:= typClimateControllerInterfaceRoom426_1.actuators.heating.setpoint;
gainHeating 				:= typClimateControllerInterfaceRoom426_1.actuators.heating.controlledVariable;

actualSetpointCooling 		:= typClimateControllerInterfaceRoom426_1.actuators.cooling.setpoint;
gainCooling 				:= typClimateControllerInterfaceRoom426_1.actuators.cooling.controlledVariable;

actualSetpointCo2			:= typClimateControllerInterfaceRoom426_1.actuators.airQuality.setpoint;
gainAirQuality				:= typClimateControllerInterfaceRoom426_1.actuators.airQuality.controlledVariable; 
damperOutput				:= typClimateControllerInterfaceRoom426_1.actuators.damper.setpoint;

currentWorkingMode			:= typClimateControllerInterfaceRoom426_1.currentMode;                   
                
                
              

ACTION settings:
                            
                                
defaultSetpoints.heating.comfort.setpoint	:= 21;
defaultSetpoints.heating.standby.setpoint	:= 2;
defaultSetpoints.heating.economy.setpoint	:= 3;
defaultSetpoints.cooling.comfort.setpoint	:= 2;
defaultSetpoints.cooling.standby.setpoint	:= 3;
defaultSetpoints.cooling.economy.setpoint	:= 4;
defaultSetpoints.co2.comfort.setpoint		:= 600;
defaultSetpoints.presenceDelayOff			:= 30;
defaultSetpoints.heating.pidSettings.KP		:= 1;
defaultSetpoints.heating.pidSettings.TN		:= 60;
defaultSetpoints.cooling.pidSettings.KP		:= 1;
defaultSetpoints.cooling.pidSettings.TN		:= 60;
defaultSetpoints.co2.pidSettings.KP			:= 20;
defaultSetpoints.co2.pidSettings.TN			:= 4000;
                            
                        
END_ACTION
END_PROGRAM

PROGRAM ClimateControl_426_2
  VAR
    climateController : FbMultiModeClimateControl_00_02;
    defaultSetpoints : typMultiModeClimateControllerDefaultSettings_00_01;
    dwConfigurationMask : DWORD := 2#0000_0000_0000_0000_0000_0001_0000_0010;
  END_VAR
  VAR_OUTPUT
    actualSetpointHeating : REAL;  (* Variabler kun for overvåking *)
    actualSetpointCooling : REAL;
    actualSetpointCo2 : REAL;
    meanTemp : REAL;
    meanCo2 : REAL;
    presence : BOOL;
    gainHeating : REAL;
    gainCooling : REAL;
    gainAirQuality : REAL;
    damperOutput : REAL;
    currentWorkingMode : enumMultiModeClimateActiveControlMode_00_01;
  END_VAR

                
    
// Innstillinger for rom:
IF (firstScan) THEN
    PersistentVars.typClimateControllerSettingsRoom426_2.ahuSystem		:= 001;
    PersistentVars.typClimateControllerSettingsRoom426_2.heatingSystem	:= 004;
    PersistentVars.typClimateControllerSettingsRoom426_2.coolingSystem	:= 004;
    defaultSetpoints 							:= PersistentVars.typClimateControlDefaultSettings;
    
// Hvis du ønsker egne innstillinger for rommet, kjør settings
    // settings();
END_IF

// Tilbakestill settpunkt (global kommando)
IF (GVL.initDefaultSettings) THEN
    climateController.setDefaultSetpoints();
END_IF

// Kjør funksjonsblokk
climateController(
    typController			:= typClimateControllerInterfaceRoom426_2, 
    typSettings				:= PersistentVars.typClimateControllerSettingsRoom426_2, 
    typDefaultSetpoints		:= defaultSetpoints,
    dwConfigurationMask		:= dwConfigurationMask            
);
        
// Registrer temperaturer
climateController.Temp          := PRG_KnxLine_1.M1_031_426_2_RMA6015_TMP_ACT.rValue_OUT;

// Registrer CO2
climateController.CO2          := PRG_KnxLine_1.M1_047_426_2_RMA6015_CO2_ACT.rValue_OUT;

// Registrer tilstedeværelse
climateController.Presence          := PRG_KnxLine_1.M1_015_426_2_RMA6015_MOV_ACT.xSwitch_OUT;

meanTemp					:= typClimateControllerInterfaceRoom426_2.actuators.heating.processValue;
meanCo2						:= climateController.Co2;
presence					:= climateController.Presence;

actualSetpointHeating 		:= typClimateControllerInterfaceRoom426_2.actuators.heating.setpoint;
gainHeating 				:= typClimateControllerInterfaceRoom426_2.actuators.heating.controlledVariable;

actualSetpointCooling 		:= typClimateControllerInterfaceRoom426_2.actuators.cooling.setpoint;
gainCooling 				:= typClimateControllerInterfaceRoom426_2.actuators.cooling.controlledVariable;

actualSetpointCo2			:= typClimateControllerInterfaceRoom426_2.actuators.airQuality.setpoint;
gainAirQuality				:= typClimateControllerInterfaceRoom426_2.actuators.airQuality.controlledVariable; 
damperOutput				:= typClimateControllerInterfaceRoom426_2.actuators.damper.setpoint;

currentWorkingMode			:= typClimateControllerInterfaceRoom426_2.currentMode;                   
                
                
              

ACTION settings:
                            
                                
defaultSetpoints.heating.comfort.setpoint	:= 21;
defaultSetpoints.heating.standby.setpoint	:= 2;
defaultSetpoints.heating.economy.setpoint	:= 3;
defaultSetpoints.cooling.comfort.setpoint	:= 2;
defaultSetpoints.cooling.standby.setpoint	:= 3;
defaultSetpoints.cooling.economy.setpoint	:= 4;
defaultSetpoints.co2.comfort.setpoint		:= 600;
defaultSetpoints.presenceDelayOff			:= 30;
defaultSetpoints.heating.pidSettings.KP		:= 1;
defaultSetpoints.heating.pidSettings.TN		:= 60;
defaultSetpoints.cooling.pidSettings.KP		:= 1;
defaultSetpoints.cooling.pidSettings.TN		:= 60;
defaultSetpoints.co2.pidSettings.KP			:= 20;
defaultSetpoints.co2.pidSettings.TN			:= 4000;
                            
                        
END_ACTION
END_PROGRAM

PROGRAM ClimateControl_426_3
  VAR
    climateController : FbMultiModeClimateControl_00_02;
    defaultSetpoints : typMultiModeClimateControllerDefaultSettings_00_01;
    dwConfigurationMask : DWORD := 2#0000_0000_0000_0000_0000_0001_0000_0010;
  END_VAR
  VAR_OUTPUT
    actualSetpointHeating : REAL;  (* Variabler kun for overvåking *)
    actualSetpointCooling : REAL;
    actualSetpointCo2 : REAL;
    meanTemp : REAL;
    meanCo2 : REAL;
    presence : BOOL;
    gainHeating : REAL;
    gainCooling : REAL;
    gainAirQuality : REAL;
    damperOutput : REAL;
    currentWorkingMode : enumMultiModeClimateActiveControlMode_00_01;
  END_VAR

                
    
// Innstillinger for rom:
IF (firstScan) THEN
    PersistentVars.typClimateControllerSettingsRoom426_3.ahuSystem		:= 001;
    PersistentVars.typClimateControllerSettingsRoom426_3.heatingSystem	:= 004;
    PersistentVars.typClimateControllerSettingsRoom426_3.coolingSystem	:= 004;
    defaultSetpoints 							:= PersistentVars.typClimateControlDefaultSettings;
    
// Hvis du ønsker egne innstillinger for rommet, kjør settings
    // settings();
END_IF

// Tilbakestill settpunkt (global kommando)
IF (GVL.initDefaultSettings) THEN
    climateController.setDefaultSetpoints();
END_IF

// Kjør funksjonsblokk
climateController(
    typController			:= typClimateControllerInterfaceRoom426_3, 
    typSettings				:= PersistentVars.typClimateControllerSettingsRoom426_3, 
    typDefaultSetpoints		:= defaultSetpoints,
    dwConfigurationMask		:= dwConfigurationMask            
);
        
// Registrer temperaturer
climateController.Temp          := PRG_KnxLine_1.M1_032_426_3_RMA6016_TMP_ACT.rValue_OUT;

// Registrer CO2
climateController.CO2          := PRG_KnxLine_1.M1_048_426_3_RMA6016_CO2_ACT.rValue_OUT;

// Registrer tilstedeværelse
climateController.Presence          := PRG_KnxLine_1.M1_016_426_3_RMA6016_MOV_ACT.xSwitch_OUT;

meanTemp					:= typClimateControllerInterfaceRoom426_3.actuators.heating.processValue;
meanCo2						:= climateController.Co2;
presence					:= climateController.Presence;

actualSetpointHeating 		:= typClimateControllerInterfaceRoom426_3.actuators.heating.setpoint;
gainHeating 				:= typClimateControllerInterfaceRoom426_3.actuators.heating.controlledVariable;

actualSetpointCooling 		:= typClimateControllerInterfaceRoom426_3.actuators.cooling.setpoint;
gainCooling 				:= typClimateControllerInterfaceRoom426_3.actuators.cooling.controlledVariable;

actualSetpointCo2			:= typClimateControllerInterfaceRoom426_3.actuators.airQuality.setpoint;
gainAirQuality				:= typClimateControllerInterfaceRoom426_3.actuators.airQuality.controlledVariable; 
damperOutput				:= typClimateControllerInterfaceRoom426_3.actuators.damper.setpoint;

currentWorkingMode			:= typClimateControllerInterfaceRoom426_3.currentMode;                   
                
                
              

ACTION settings:
                            
                                
defaultSetpoints.heating.comfort.setpoint	:= 21;
defaultSetpoints.heating.standby.setpoint	:= 2;
defaultSetpoints.heating.economy.setpoint	:= 3;
defaultSetpoints.cooling.comfort.setpoint	:= 2;
defaultSetpoints.cooling.standby.setpoint	:= 3;
defaultSetpoints.cooling.economy.setpoint	:= 4;
defaultSetpoints.co2.comfort.setpoint		:= 600;
defaultSetpoints.presenceDelayOff			:= 30;
defaultSetpoints.heating.pidSettings.KP		:= 1;
defaultSetpoints.heating.pidSettings.TN		:= 60;
defaultSetpoints.cooling.pidSettings.KP		:= 1;
defaultSetpoints.cooling.pidSettings.TN		:= 60;
defaultSetpoints.co2.pidSettings.KP			:= 20;
defaultSetpoints.co2.pidSettings.TN			:= 4000;
                            
                        
END_ACTION
END_PROGRAM

PROGRAM ClimateControl_528
  VAR
    climateController : FbMultiModeClimateControl_00_02;
    defaultSetpoints : typMultiModeClimateControllerDefaultSettings_00_01;
    dwConfigurationMask : DWORD := 2#0000_0000_0000_0000_0000_0001_0000_0010;
  END_VAR
  VAR_OUTPUT
    actualSetpointHeating : REAL;  (* Variabler kun for overvåking *)
    actualSetpointCooling : REAL;
    actualSetpointCo2 : REAL;
    meanTemp : REAL;
    meanCo2 : REAL;
    presence : BOOL;
    gainHeating : REAL;
    gainCooling : REAL;
    gainAirQuality : REAL;
    damperOutput : REAL;
    currentWorkingMode : enumMultiModeClimateActiveControlMode_00_01;
  END_VAR

                
    
// Innstillinger for rom:
IF (firstScan) THEN
    PersistentVars.typClimateControllerSettingsRoom528.ahuSystem		:= 001;
    PersistentVars.typClimateControllerSettingsRoom528.heatingSystem	:= 005;
    PersistentVars.typClimateControllerSettingsRoom528.coolingSystem	:= 005;
    defaultSetpoints 							:= PersistentVars.typClimateControlDefaultSettings;
    
// Hvis du ønsker egne innstillinger for rommet, kjør settings
    // settings();
END_IF

// Tilbakestill settpunkt (global kommando)
IF (GVL.initDefaultSettings) THEN
    climateController.setDefaultSetpoints();
END_IF

// Kjør funksjonsblokk
climateController(
    typController			:= typClimateControllerInterfaceRoom528, 
    typSettings				:= PersistentVars.typClimateControllerSettingsRoom528, 
    typDefaultSetpoints		:= defaultSetpoints,
    dwConfigurationMask		:= dwConfigurationMask            
);
        
// Registrer temperaturer
climateController.Temp          := PRG_KnxLine_2.M2_013_528_RMA6001_TMP_ACT.rValue_OUT;

// Registrer CO2
climateController.CO2          := PRG_KnxLine_2.M2_025_528_RMA6001_CO2_ACT.rValue_OUT;

// Registrer tilstedeværelse
climateController.Presence          := PRG_KnxLine_2.M2_001_528_RMA6001_MOV_ACT.xSwitch_OUT;

meanTemp					:= typClimateControllerInterfaceRoom528.actuators.heating.processValue;
meanCo2						:= climateController.Co2;
presence					:= climateController.Presence;

actualSetpointHeating 		:= typClimateControllerInterfaceRoom528.actuators.heating.setpoint;
gainHeating 				:= typClimateControllerInterfaceRoom528.actuators.heating.controlledVariable;

actualSetpointCooling 		:= typClimateControllerInterfaceRoom528.actuators.cooling.setpoint;
gainCooling 				:= typClimateControllerInterfaceRoom528.actuators.cooling.controlledVariable;

actualSetpointCo2			:= typClimateControllerInterfaceRoom528.actuators.airQuality.setpoint;
gainAirQuality				:= typClimateControllerInterfaceRoom528.actuators.airQuality.controlledVariable; 
damperOutput				:= typClimateControllerInterfaceRoom528.actuators.damper.setpoint;

currentWorkingMode			:= typClimateControllerInterfaceRoom528.currentMode;                   
                
                
              

ACTION settings:
                            
                                
defaultSetpoints.heating.comfort.setpoint	:= 21;
defaultSetpoints.heating.standby.setpoint	:= 2;
defaultSetpoints.heating.economy.setpoint	:= 3;
defaultSetpoints.cooling.comfort.setpoint	:= 2;
defaultSetpoints.cooling.standby.setpoint	:= 3;
defaultSetpoints.cooling.economy.setpoint	:= 4;
defaultSetpoints.co2.comfort.setpoint		:= 600;
defaultSetpoints.presenceDelayOff			:= 30;
defaultSetpoints.heating.pidSettings.KP		:= 1;
defaultSetpoints.heating.pidSettings.TN		:= 60;
defaultSetpoints.cooling.pidSettings.KP		:= 1;
defaultSetpoints.cooling.pidSettings.TN		:= 60;
defaultSetpoints.co2.pidSettings.KP			:= 20;
defaultSetpoints.co2.pidSettings.TN			:= 4000;
                            
                        
END_ACTION
END_PROGRAM

PROGRAM ClimateControl_523
  VAR
    climateController : FbMultiModeClimateControl_00_02;
    defaultSetpoints : typMultiModeClimateControllerDefaultSettings_00_01;
    dwConfigurationMask : DWORD := 2#0000_0000_0000_0000_0000_0001_0000_0010;
  END_VAR
  VAR_OUTPUT
    actualSetpointHeating : REAL;  (* Variabler kun for overvåking *)
    actualSetpointCooling : REAL;
    actualSetpointCo2 : REAL;
    meanTemp : REAL;
    meanCo2 : REAL;
    presence : BOOL;
    gainHeating : REAL;
    gainCooling : REAL;
    gainAirQuality : REAL;
    damperOutput : REAL;
    currentWorkingMode : enumMultiModeClimateActiveControlMode_00_01;
  END_VAR

                
    
// Innstillinger for rom:
IF (firstScan) THEN
    PersistentVars.typClimateControllerSettingsRoom523.ahuSystem		:= 001;
    PersistentVars.typClimateControllerSettingsRoom523.heatingSystem	:= 005;
    PersistentVars.typClimateControllerSettingsRoom523.coolingSystem	:= 005;
    defaultSetpoints 							:= PersistentVars.typClimateControlDefaultSettings;
    
// Hvis du ønsker egne innstillinger for rommet, kjør settings
    // settings();
END_IF

// Tilbakestill settpunkt (global kommando)
IF (GVL.initDefaultSettings) THEN
    climateController.setDefaultSetpoints();
END_IF

// Kjør funksjonsblokk
climateController(
    typController			:= typClimateControllerInterfaceRoom523, 
    typSettings				:= PersistentVars.typClimateControllerSettingsRoom523, 
    typDefaultSetpoints		:= defaultSetpoints,
    dwConfigurationMask		:= dwConfigurationMask            
);
        
// Registrer temperaturer
climateController.Temp          := PRG_KnxLine_2.M2_014_523_RMA6002_TMP_ACT.rValue_OUT;

// Registrer CO2
climateController.CO2          := PRG_KnxLine_2.M2_026_523_RMA6002_CO2_ACT.rValue_OUT;

// Registrer tilstedeværelse
climateController.Presence          := PRG_KnxLine_2.M2_002_523_RMA6002_MOV_ACT.xSwitch_OUT;

meanTemp					:= typClimateControllerInterfaceRoom523.actuators.heating.processValue;
meanCo2						:= climateController.Co2;
presence					:= climateController.Presence;

actualSetpointHeating 		:= typClimateControllerInterfaceRoom523.actuators.heating.setpoint;
gainHeating 				:= typClimateControllerInterfaceRoom523.actuators.heating.controlledVariable;

actualSetpointCooling 		:= typClimateControllerInterfaceRoom523.actuators.cooling.setpoint;
gainCooling 				:= typClimateControllerInterfaceRoom523.actuators.cooling.controlledVariable;

actualSetpointCo2			:= typClimateControllerInterfaceRoom523.actuators.airQuality.setpoint;
gainAirQuality				:= typClimateControllerInterfaceRoom523.actuators.airQuality.controlledVariable; 
damperOutput				:= typClimateControllerInterfaceRoom523.actuators.damper.setpoint;

currentWorkingMode			:= typClimateControllerInterfaceRoom523.currentMode;                   
                
                
              

ACTION settings:
                            
                                
defaultSetpoints.heating.comfort.setpoint	:= 21;
defaultSetpoints.heating.standby.setpoint	:= 2;
defaultSetpoints.heating.economy.setpoint	:= 3;
defaultSetpoints.cooling.comfort.setpoint	:= 2;
defaultSetpoints.cooling.standby.setpoint	:= 3;
defaultSetpoints.cooling.economy.setpoint	:= 4;
defaultSetpoints.co2.comfort.setpoint		:= 600;
defaultSetpoints.presenceDelayOff			:= 30;
defaultSetpoints.heating.pidSettings.KP		:= 1;
defaultSetpoints.heating.pidSettings.TN		:= 60;
defaultSetpoints.cooling.pidSettings.KP		:= 1;
defaultSetpoints.cooling.pidSettings.TN		:= 60;
defaultSetpoints.co2.pidSettings.KP			:= 20;
defaultSetpoints.co2.pidSettings.TN			:= 4000;
                            
                        
END_ACTION
END_PROGRAM

PROGRAM ClimateControl_531
  VAR
    climateController : FbMultiModeClimateControl_00_02;
    defaultSetpoints : typMultiModeClimateControllerDefaultSettings_00_01;
    dwConfigurationMask : DWORD := 2#0000_0000_0000_0000_0000_0001_0000_0010;
  END_VAR
  VAR_OUTPUT
    actualSetpointHeating : REAL;  (* Variabler kun for overvåking *)
    actualSetpointCooling : REAL;
    actualSetpointCo2 : REAL;
    meanTemp : REAL;
    meanCo2 : REAL;
    presence : BOOL;
    gainHeating : REAL;
    gainCooling : REAL;
    gainAirQuality : REAL;
    damperOutput : REAL;
    currentWorkingMode : enumMultiModeClimateActiveControlMode_00_01;
  END_VAR

                
    
// Innstillinger for rom:
IF (firstScan) THEN
    PersistentVars.typClimateControllerSettingsRoom531.ahuSystem		:= 001;
    PersistentVars.typClimateControllerSettingsRoom531.heatingSystem	:= 005;
    PersistentVars.typClimateControllerSettingsRoom531.coolingSystem	:= 005;
    defaultSetpoints 							:= PersistentVars.typClimateControlDefaultSettings;
    
// Hvis du ønsker egne innstillinger for rommet, kjør settings
    // settings();
END_IF

// Tilbakestill settpunkt (global kommando)
IF (GVL.initDefaultSettings) THEN
    climateController.setDefaultSetpoints();
END_IF

// Kjør funksjonsblokk
climateController(
    typController			:= typClimateControllerInterfaceRoom531, 
    typSettings				:= PersistentVars.typClimateControllerSettingsRoom531, 
    typDefaultSetpoints		:= defaultSetpoints,
    dwConfigurationMask		:= dwConfigurationMask            
);
        
// Registrer temperaturer
climateController.Temp          := PRG_KnxLine_2.M2_015_531_RMA6003_TMP_ACT.rValue_OUT;

// Registrer CO2
climateController.CO2          := PRG_KnxLine_2.M2_027_531_RMA6003_CO2_ACT.rValue_OUT;

// Registrer tilstedeværelse
climateController.Presence          := PRG_KnxLine_2.M2_003_531_RMA6003_MOV_ACT.xSwitch_OUT;

meanTemp					:= typClimateControllerInterfaceRoom531.actuators.heating.processValue;
meanCo2						:= climateController.Co2;
presence					:= climateController.Presence;

actualSetpointHeating 		:= typClimateControllerInterfaceRoom531.actuators.heating.setpoint;
gainHeating 				:= typClimateControllerInterfaceRoom531.actuators.heating.controlledVariable;

actualSetpointCooling 		:= typClimateControllerInterfaceRoom531.actuators.cooling.setpoint;
gainCooling 				:= typClimateControllerInterfaceRoom531.actuators.cooling.controlledVariable;

actualSetpointCo2			:= typClimateControllerInterfaceRoom531.actuators.airQuality.setpoint;
gainAirQuality				:= typClimateControllerInterfaceRoom531.actuators.airQuality.controlledVariable; 
damperOutput				:= typClimateControllerInterfaceRoom531.actuators.damper.setpoint;

currentWorkingMode			:= typClimateControllerInterfaceRoom531.currentMode;                   
                
                
              

ACTION settings:
                            
                                
defaultSetpoints.heating.comfort.setpoint	:= 21;
defaultSetpoints.heating.standby.setpoint	:= 2;
defaultSetpoints.heating.economy.setpoint	:= 3;
defaultSetpoints.cooling.comfort.setpoint	:= 2;
defaultSetpoints.cooling.standby.setpoint	:= 3;
defaultSetpoints.cooling.economy.setpoint	:= 4;
defaultSetpoints.co2.comfort.setpoint		:= 600;
defaultSetpoints.presenceDelayOff			:= 30;
defaultSetpoints.heating.pidSettings.KP		:= 1;
defaultSetpoints.heating.pidSettings.TN		:= 60;
defaultSetpoints.cooling.pidSettings.KP		:= 1;
defaultSetpoints.cooling.pidSettings.TN		:= 60;
defaultSetpoints.co2.pidSettings.KP			:= 20;
defaultSetpoints.co2.pidSettings.TN			:= 4000;
                            
                        
END_ACTION
END_PROGRAM

PROGRAM ClimateControl_535_1
  VAR
    climateController : FbMultiModeClimateControl_00_02;
    defaultSetpoints : typMultiModeClimateControllerDefaultSettings_00_01;
    dwConfigurationMask : DWORD := 2#0000_0000_0000_0000_0000_0001_0000_0010;
  END_VAR
  VAR_OUTPUT
    actualSetpointHeating : REAL;  (* Variabler kun for overvåking *)
    actualSetpointCooling : REAL;
    actualSetpointCo2 : REAL;
    meanTemp : REAL;
    meanCo2 : REAL;
    presence : BOOL;
    gainHeating : REAL;
    gainCooling : REAL;
    gainAirQuality : REAL;
    damperOutput : REAL;
    currentWorkingMode : enumMultiModeClimateActiveControlMode_00_01;
  END_VAR

                
    
// Innstillinger for rom:
IF (firstScan) THEN
    PersistentVars.typClimateControllerSettingsRoom535_1.ahuSystem		:= 001;
    PersistentVars.typClimateControllerSettingsRoom535_1.heatingSystem	:= 005;
    PersistentVars.typClimateControllerSettingsRoom535_1.coolingSystem	:= 005;
    defaultSetpoints 							:= PersistentVars.typClimateControlDefaultSettings;
    
// Hvis du ønsker egne innstillinger for rommet, kjør settings
    // settings();
END_IF

// Tilbakestill settpunkt (global kommando)
IF (GVL.initDefaultSettings) THEN
    climateController.setDefaultSetpoints();
END_IF

// Kjør funksjonsblokk
climateController(
    typController			:= typClimateControllerInterfaceRoom535_1, 
    typSettings				:= PersistentVars.typClimateControllerSettingsRoom535_1, 
    typDefaultSetpoints		:= defaultSetpoints,
    dwConfigurationMask		:= dwConfigurationMask            
);
        
// Registrer temperaturer
climateController.Temp          := PRG_KnxLine_2.M2_016_535_1_RMA6004_TMP_ACT.rValue_OUT;

// Registrer CO2
climateController.CO2          := PRG_KnxLine_2.M2_028_535_1_RMA6004_CO2_ACT.rValue_OUT;

// Registrer tilstedeværelse
climateController.Presence          := PRG_KnxLine_2.M2_004_535_1_RMA6004_MOV_ACT.xSwitch_OUT;

meanTemp					:= typClimateControllerInterfaceRoom535_1.actuators.heating.processValue;
meanCo2						:= climateController.Co2;
presence					:= climateController.Presence;

actualSetpointHeating 		:= typClimateControllerInterfaceRoom535_1.actuators.heating.setpoint;
gainHeating 				:= typClimateControllerInterfaceRoom535_1.actuators.heating.controlledVariable;

actualSetpointCooling 		:= typClimateControllerInterfaceRoom535_1.actuators.cooling.setpoint;
gainCooling 				:= typClimateControllerInterfaceRoom535_1.actuators.cooling.controlledVariable;

actualSetpointCo2			:= typClimateControllerInterfaceRoom535_1.actuators.airQuality.setpoint;
gainAirQuality				:= typClimateControllerInterfaceRoom535_1.actuators.airQuality.controlledVariable; 
damperOutput				:= typClimateControllerInterfaceRoom535_1.actuators.damper.setpoint;

currentWorkingMode			:= typClimateControllerInterfaceRoom535_1.currentMode;                   
                
                
              

ACTION settings:
                            
                                
defaultSetpoints.heating.comfort.setpoint	:= 21;
defaultSetpoints.heating.standby.setpoint	:= 2;
defaultSetpoints.heating.economy.setpoint	:= 3;
defaultSetpoints.cooling.comfort.setpoint	:= 2;
defaultSetpoints.cooling.standby.setpoint	:= 3;
defaultSetpoints.cooling.economy.setpoint	:= 4;
defaultSetpoints.co2.comfort.setpoint		:= 600;
defaultSetpoints.presenceDelayOff			:= 30;
defaultSetpoints.heating.pidSettings.KP		:= 1;
defaultSetpoints.heating.pidSettings.TN		:= 60;
defaultSetpoints.cooling.pidSettings.KP		:= 1;
defaultSetpoints.cooling.pidSettings.TN		:= 60;
defaultSetpoints.co2.pidSettings.KP			:= 20;
defaultSetpoints.co2.pidSettings.TN			:= 4000;
                            
                        
END_ACTION
END_PROGRAM

PROGRAM ClimateControl_535_2
  VAR
    climateController : FbMultiModeClimateControl_00_02;
    defaultSetpoints : typMultiModeClimateControllerDefaultSettings_00_01;
    dwConfigurationMask : DWORD := 2#0000_0000_0000_0000_0000_0001_0000_0010;
  END_VAR
  VAR_OUTPUT
    actualSetpointHeating : REAL;  (* Variabler kun for overvåking *)
    actualSetpointCooling : REAL;
    actualSetpointCo2 : REAL;
    meanTemp : REAL;
    meanCo2 : REAL;
    presence : BOOL;
    gainHeating : REAL;
    gainCooling : REAL;
    gainAirQuality : REAL;
    damperOutput : REAL;
    currentWorkingMode : enumMultiModeClimateActiveControlMode_00_01;
  END_VAR

                
    
// Innstillinger for rom:
IF (firstScan) THEN
    PersistentVars.typClimateControllerSettingsRoom535_2.ahuSystem		:= 001;
    PersistentVars.typClimateControllerSettingsRoom535_2.heatingSystem	:= 005;
    PersistentVars.typClimateControllerSettingsRoom535_2.coolingSystem	:= 005;
    defaultSetpoints 							:= PersistentVars.typClimateControlDefaultSettings;
    
// Hvis du ønsker egne innstillinger for rommet, kjør settings
    // settings();
END_IF

// Tilbakestill settpunkt (global kommando)
IF (GVL.initDefaultSettings) THEN
    climateController.setDefaultSetpoints();
END_IF

// Kjør funksjonsblokk
climateController(
    typController			:= typClimateControllerInterfaceRoom535_2, 
    typSettings				:= PersistentVars.typClimateControllerSettingsRoom535_2, 
    typDefaultSetpoints		:= defaultSetpoints,
    dwConfigurationMask		:= dwConfigurationMask            
);
        
// Registrer temperaturer
climateController.Temp          := PRG_KnxLine_2.M2_017_535_2_RMA6005_TMP_ACT.rValue_OUT;

// Registrer CO2
climateController.CO2          := PRG_KnxLine_2.M2_029_535_2_RMA6005_CO2_ACT.rValue_OUT;

// Registrer tilstedeværelse
climateController.Presence          := PRG_KnxLine_2.M2_005_535_2_RMA6005_MOV_ACT.xSwitch_OUT;

meanTemp					:= typClimateControllerInterfaceRoom535_2.actuators.heating.processValue;
meanCo2						:= climateController.Co2;
presence					:= climateController.Presence;

actualSetpointHeating 		:= typClimateControllerInterfaceRoom535_2.actuators.heating.setpoint;
gainHeating 				:= typClimateControllerInterfaceRoom535_2.actuators.heating.controlledVariable;

actualSetpointCooling 		:= typClimateControllerInterfaceRoom535_2.actuators.cooling.setpoint;
gainCooling 				:= typClimateControllerInterfaceRoom535_2.actuators.cooling.controlledVariable;

actualSetpointCo2			:= typClimateControllerInterfaceRoom535_2.actuators.airQuality.setpoint;
gainAirQuality				:= typClimateControllerInterfaceRoom535_2.actuators.airQuality.controlledVariable; 
damperOutput				:= typClimateControllerInterfaceRoom535_2.actuators.damper.setpoint;

currentWorkingMode			:= typClimateControllerInterfaceRoom535_2.currentMode;                   
                
                
              

ACTION settings:
                            
                                
defaultSetpoints.heating.comfort.setpoint	:= 21;
defaultSetpoints.heating.standby.setpoint	:= 2;
defaultSetpoints.heating.economy.setpoint	:= 3;
defaultSetpoints.cooling.comfort.setpoint	:= 2;
defaultSetpoints.cooling.standby.setpoint	:= 3;
defaultSetpoints.cooling.economy.setpoint	:= 4;
defaultSetpoints.co2.comfort.setpoint		:= 600;
defaultSetpoints.presenceDelayOff			:= 30;
defaultSetpoints.heating.pidSettings.KP		:= 1;
defaultSetpoints.heating.pidSettings.TN		:= 60;
defaultSetpoints.cooling.pidSettings.KP		:= 1;
defaultSetpoints.cooling.pidSettings.TN		:= 60;
defaultSetpoints.co2.pidSettings.KP			:= 20;
defaultSetpoints.co2.pidSettings.TN			:= 4000;
                            
                        
END_ACTION
END_PROGRAM

PROGRAM ClimateControl_535_3
  VAR
    climateController : FbMultiModeClimateControl_00_02;
    defaultSetpoints : typMultiModeClimateControllerDefaultSettings_00_01;
    dwConfigurationMask : DWORD := 2#0000_0000_0000_0000_0000_0001_0000_0010;
  END_VAR
  VAR_OUTPUT
    actualSetpointHeating : REAL;  (* Variabler kun for overvåking *)
    actualSetpointCooling : REAL;
    actualSetpointCo2 : REAL;
    meanTemp : REAL;
    meanCo2 : REAL;
    presence : BOOL;
    gainHeating : REAL;
    gainCooling : REAL;
    gainAirQuality : REAL;
    damperOutput : REAL;
    currentWorkingMode : enumMultiModeClimateActiveControlMode_00_01;
  END_VAR

                
    
// Innstillinger for rom:
IF (firstScan) THEN
    PersistentVars.typClimateControllerSettingsRoom535_3.ahuSystem		:= 001;
    PersistentVars.typClimateControllerSettingsRoom535_3.heatingSystem	:= 005;
    PersistentVars.typClimateControllerSettingsRoom535_3.coolingSystem	:= 005;
    defaultSetpoints 							:= PersistentVars.typClimateControlDefaultSettings;
    
// Hvis du ønsker egne innstillinger for rommet, kjør settings
    // settings();
END_IF

// Tilbakestill settpunkt (global kommando)
IF (GVL.initDefaultSettings) THEN
    climateController.setDefaultSetpoints();
END_IF

// Kjør funksjonsblokk
climateController(
    typController			:= typClimateControllerInterfaceRoom535_3, 
    typSettings				:= PersistentVars.typClimateControllerSettingsRoom535_3, 
    typDefaultSetpoints		:= defaultSetpoints,
    dwConfigurationMask		:= dwConfigurationMask            
);
        
// Registrer temperaturer
climateController.Temp          := PRG_KnxLine_2.M2_018_535_3_RMA6006_TMP_ACT.rValue_OUT;

// Registrer CO2
climateController.CO2          := PRG_KnxLine_2.M2_030_535_3_RMA6006_CO2_ACT.rValue_OUT;

// Registrer tilstedeværelse
climateController.Presence          := PRG_KnxLine_2.M2_006_535_3_RMA6006_MOV_ACT.xSwitch_OUT;

meanTemp					:= typClimateControllerInterfaceRoom535_3.actuators.heating.processValue;
meanCo2						:= climateController.Co2;
presence					:= climateController.Presence;

actualSetpointHeating 		:= typClimateControllerInterfaceRoom535_3.actuators.heating.setpoint;
gainHeating 				:= typClimateControllerInterfaceRoom535_3.actuators.heating.controlledVariable;

actualSetpointCooling 		:= typClimateControllerInterfaceRoom535_3.actuators.cooling.setpoint;
gainCooling 				:= typClimateControllerInterfaceRoom535_3.actuators.cooling.controlledVariable;

actualSetpointCo2			:= typClimateControllerInterfaceRoom535_3.actuators.airQuality.setpoint;
gainAirQuality				:= typClimateControllerInterfaceRoom535_3.actuators.airQuality.controlledVariable; 
damperOutput				:= typClimateControllerInterfaceRoom535_3.actuators.damper.setpoint;

currentWorkingMode			:= typClimateControllerInterfaceRoom535_3.currentMode;                   
                
                
              

ACTION settings:
                            
                                
defaultSetpoints.heating.comfort.setpoint	:= 21;
defaultSetpoints.heating.standby.setpoint	:= 2;
defaultSetpoints.heating.economy.setpoint	:= 3;
defaultSetpoints.cooling.comfort.setpoint	:= 2;
defaultSetpoints.cooling.standby.setpoint	:= 3;
defaultSetpoints.cooling.economy.setpoint	:= 4;
defaultSetpoints.co2.comfort.setpoint		:= 600;
defaultSetpoints.presenceDelayOff			:= 30;
defaultSetpoints.heating.pidSettings.KP		:= 1;
defaultSetpoints.heating.pidSettings.TN		:= 60;
defaultSetpoints.cooling.pidSettings.KP		:= 1;
defaultSetpoints.cooling.pidSettings.TN		:= 60;
defaultSetpoints.co2.pidSettings.KP			:= 20;
defaultSetpoints.co2.pidSettings.TN			:= 4000;
                            
                        
END_ACTION
END_PROGRAM

PROGRAM ClimateControl_536
  VAR
    climateController : FbMultiModeClimateControl_00_02;
    defaultSetpoints : typMultiModeClimateControllerDefaultSettings_00_01;
    dwConfigurationMask : DWORD := 2#0000_0000_0000_0000_0000_0001_0000_0010;
  END_VAR
  VAR_OUTPUT
    actualSetpointHeating : REAL;  (* Variabler kun for overvåking *)
    actualSetpointCooling : REAL;
    actualSetpointCo2 : REAL;
    meanTemp : REAL;
    meanCo2 : REAL;
    presence : BOOL;
    gainHeating : REAL;
    gainCooling : REAL;
    gainAirQuality : REAL;
    damperOutput : REAL;
    currentWorkingMode : enumMultiModeClimateActiveControlMode_00_01;
  END_VAR

                
    
// Innstillinger for rom:
IF (firstScan) THEN
    PersistentVars.typClimateControllerSettingsRoom536.ahuSystem		:= 001;
    PersistentVars.typClimateControllerSettingsRoom536.heatingSystem	:= 005;
    PersistentVars.typClimateControllerSettingsRoom536.coolingSystem	:= 005;
    defaultSetpoints 							:= PersistentVars.typClimateControlDefaultSettings;
    
// Hvis du ønsker egne innstillinger for rommet, kjør settings
    // settings();
END_IF

// Tilbakestill settpunkt (global kommando)
IF (GVL.initDefaultSettings) THEN
    climateController.setDefaultSetpoints();
END_IF

// Kjør funksjonsblokk
climateController(
    typController			:= typClimateControllerInterfaceRoom536, 
    typSettings				:= PersistentVars.typClimateControllerSettingsRoom536, 
    typDefaultSetpoints		:= defaultSetpoints,
    dwConfigurationMask		:= dwConfigurationMask            
);
        
// Registrer temperaturer
climateController.Temp          := PRG_KnxLine_2.M2_019_536_RMA6007_TMP_ACT.rValue_OUT;

// Registrer CO2
climateController.CO2          := PRG_KnxLine_2.M2_031_536_RMA6007_CO2_ACT.rValue_OUT;

// Registrer tilstedeværelse
climateController.Presence          := PRG_KnxLine_2.M2_007_536_RMA6007_MOV_ACT.xSwitch_OUT;

meanTemp					:= typClimateControllerInterfaceRoom536.actuators.heating.processValue;
meanCo2						:= climateController.Co2;
presence					:= climateController.Presence;

actualSetpointHeating 		:= typClimateControllerInterfaceRoom536.actuators.heating.setpoint;
gainHeating 				:= typClimateControllerInterfaceRoom536.actuators.heating.controlledVariable;

actualSetpointCooling 		:= typClimateControllerInterfaceRoom536.actuators.cooling.setpoint;
gainCooling 				:= typClimateControllerInterfaceRoom536.actuators.cooling.controlledVariable;

actualSetpointCo2			:= typClimateControllerInterfaceRoom536.actuators.airQuality.setpoint;
gainAirQuality				:= typClimateControllerInterfaceRoom536.actuators.airQuality.controlledVariable; 
damperOutput				:= typClimateControllerInterfaceRoom536.actuators.damper.setpoint;

currentWorkingMode			:= typClimateControllerInterfaceRoom536.currentMode;                   
                
                
              

ACTION settings:
                            
                                
defaultSetpoints.heating.comfort.setpoint	:= 21;
defaultSetpoints.heating.standby.setpoint	:= 2;
defaultSetpoints.heating.economy.setpoint	:= 3;
defaultSetpoints.cooling.comfort.setpoint	:= 2;
defaultSetpoints.cooling.standby.setpoint	:= 3;
defaultSetpoints.cooling.economy.setpoint	:= 4;
defaultSetpoints.co2.comfort.setpoint		:= 600;
defaultSetpoints.presenceDelayOff			:= 30;
defaultSetpoints.heating.pidSettings.KP		:= 1;
defaultSetpoints.heating.pidSettings.TN		:= 60;
defaultSetpoints.cooling.pidSettings.KP		:= 1;
defaultSetpoints.cooling.pidSettings.TN		:= 60;
defaultSetpoints.co2.pidSettings.KP			:= 20;
defaultSetpoints.co2.pidSettings.TN			:= 4000;
                            
                        
END_ACTION
END_PROGRAM

PROGRAM ClimateControl_543
  VAR
    climateController : FbMultiModeClimateControl_00_02;
    defaultSetpoints : typMultiModeClimateControllerDefaultSettings_00_01;
    dwConfigurationMask : DWORD := 2#0000_0000_0000_0000_0000_0001_0000_0010;
  END_VAR
  VAR_OUTPUT
    actualSetpointHeating : REAL;  (* Variabler kun for overvåking *)
    actualSetpointCooling : REAL;
    actualSetpointCo2 : REAL;
    meanTemp : REAL;
    meanCo2 : REAL;
    presence : BOOL;
    gainHeating : REAL;
    gainCooling : REAL;
    gainAirQuality : REAL;
    damperOutput : REAL;
    currentWorkingMode : enumMultiModeClimateActiveControlMode_00_01;
  END_VAR

                
    
// Innstillinger for rom:
IF (firstScan) THEN
    PersistentVars.typClimateControllerSettingsRoom543.ahuSystem		:= 001;
    PersistentVars.typClimateControllerSettingsRoom543.heatingSystem	:= 005;
    PersistentVars.typClimateControllerSettingsRoom543.coolingSystem	:= 005;
    defaultSetpoints 							:= PersistentVars.typClimateControlDefaultSettings;
    
// Hvis du ønsker egne innstillinger for rommet, kjør settings
    // settings();
END_IF

// Tilbakestill settpunkt (global kommando)
IF (GVL.initDefaultSettings) THEN
    climateController.setDefaultSetpoints();
END_IF

// Kjør funksjonsblokk
climateController(
    typController			:= typClimateControllerInterfaceRoom543, 
    typSettings				:= PersistentVars.typClimateControllerSettingsRoom543, 
    typDefaultSetpoints		:= defaultSetpoints,
    dwConfigurationMask		:= dwConfigurationMask            
);
        
// Registrer temperaturer
climateController.Temp          := PRG_KnxLine_2.M2_020_543_RMA6008_TMP_ACT.rValue_OUT;

// Registrer CO2
climateController.CO2          := PRG_KnxLine_2.M2_032_543_RMA6008_CO2_ACT.rValue_OUT;

// Registrer tilstedeværelse
climateController.Presence          := PRG_KnxLine_2.M2_008_543_RMA6008_MOV_ACT.xSwitch_OUT;

meanTemp					:= typClimateControllerInterfaceRoom543.actuators.heating.processValue;
meanCo2						:= climateController.Co2;
presence					:= climateController.Presence;

actualSetpointHeating 		:= typClimateControllerInterfaceRoom543.actuators.heating.setpoint;
gainHeating 				:= typClimateControllerInterfaceRoom543.actuators.heating.controlledVariable;

actualSetpointCooling 		:= typClimateControllerInterfaceRoom543.actuators.cooling.setpoint;
gainCooling 				:= typClimateControllerInterfaceRoom543.actuators.cooling.controlledVariable;

actualSetpointCo2			:= typClimateControllerInterfaceRoom543.actuators.airQuality.setpoint;
gainAirQuality				:= typClimateControllerInterfaceRoom543.actuators.airQuality.controlledVariable; 
damperOutput				:= typClimateControllerInterfaceRoom543.actuators.damper.setpoint;

currentWorkingMode			:= typClimateControllerInterfaceRoom543.currentMode;                   
                
                
              

ACTION settings:
                            
                                
defaultSetpoints.heating.comfort.setpoint	:= 21;
defaultSetpoints.heating.standby.setpoint	:= 2;
defaultSetpoints.heating.economy.setpoint	:= 3;
defaultSetpoints.cooling.comfort.setpoint	:= 2;
defaultSetpoints.cooling.standby.setpoint	:= 3;
defaultSetpoints.cooling.economy.setpoint	:= 4;
defaultSetpoints.co2.comfort.setpoint		:= 600;
defaultSetpoints.presenceDelayOff			:= 30;
defaultSetpoints.heating.pidSettings.KP		:= 1;
defaultSetpoints.heating.pidSettings.TN		:= 60;
defaultSetpoints.cooling.pidSettings.KP		:= 1;
defaultSetpoints.cooling.pidSettings.TN		:= 60;
defaultSetpoints.co2.pidSettings.KP			:= 20;
defaultSetpoints.co2.pidSettings.TN			:= 4000;
                            
                        
END_ACTION
END_PROGRAM

PROGRAM ClimateControl_547_1
  VAR
    climateController : FbMultiModeClimateControl_00_02;
    defaultSetpoints : typMultiModeClimateControllerDefaultSettings_00_01;
    dwConfigurationMask : DWORD := 2#0000_0000_0000_0000_0000_0001_0000_0010;
  END_VAR
  VAR_OUTPUT
    actualSetpointHeating : REAL;  (* Variabler kun for overvåking *)
    actualSetpointCooling : REAL;
    actualSetpointCo2 : REAL;
    meanTemp : REAL;
    meanCo2 : REAL;
    presence : BOOL;
    gainHeating : REAL;
    gainCooling : REAL;
    gainAirQuality : REAL;
    damperOutput : REAL;
    currentWorkingMode : enumMultiModeClimateActiveControlMode_00_01;
  END_VAR

                
    
// Innstillinger for rom:
IF (firstScan) THEN
    PersistentVars.typClimateControllerSettingsRoom547_1.ahuSystem		:= 001;
    PersistentVars.typClimateControllerSettingsRoom547_1.heatingSystem	:= 005;
    PersistentVars.typClimateControllerSettingsRoom547_1.coolingSystem	:= 005;
    defaultSetpoints 							:= PersistentVars.typClimateControlDefaultSettings;
    
// Hvis du ønsker egne innstillinger for rommet, kjør settings
    // settings();
END_IF

// Tilbakestill settpunkt (global kommando)
IF (GVL.initDefaultSettings) THEN
    climateController.setDefaultSetpoints();
END_IF

// Kjør funksjonsblokk
climateController(
    typController			:= typClimateControllerInterfaceRoom547_1, 
    typSettings				:= PersistentVars.typClimateControllerSettingsRoom547_1, 
    typDefaultSetpoints		:= defaultSetpoints,
    dwConfigurationMask		:= dwConfigurationMask            
);
        
// Registrer temperaturer
climateController.Temp          := PRG_KnxLine_2.M2_021_547_1_RMA6009_TMP_ACT.rValue_OUT;

// Registrer CO2
climateController.CO2          := PRG_KnxLine_2.M2_033_547_1_RMA6009_CO2_ACT.rValue_OUT;

// Registrer tilstedeværelse
climateController.Presence          := PRG_KnxLine_2.M2_009_547_1_RMA6009_MOV_ACT.xSwitch_OUT;

meanTemp					:= typClimateControllerInterfaceRoom547_1.actuators.heating.processValue;
meanCo2						:= climateController.Co2;
presence					:= climateController.Presence;

actualSetpointHeating 		:= typClimateControllerInterfaceRoom547_1.actuators.heating.setpoint;
gainHeating 				:= typClimateControllerInterfaceRoom547_1.actuators.heating.controlledVariable;

actualSetpointCooling 		:= typClimateControllerInterfaceRoom547_1.actuators.cooling.setpoint;
gainCooling 				:= typClimateControllerInterfaceRoom547_1.actuators.cooling.controlledVariable;

actualSetpointCo2			:= typClimateControllerInterfaceRoom547_1.actuators.airQuality.setpoint;
gainAirQuality				:= typClimateControllerInterfaceRoom547_1.actuators.airQuality.controlledVariable; 
damperOutput				:= typClimateControllerInterfaceRoom547_1.actuators.damper.setpoint;

currentWorkingMode			:= typClimateControllerInterfaceRoom547_1.currentMode;                   
                
                
              

ACTION settings:
                            
                                
defaultSetpoints.heating.comfort.setpoint	:= 21;
defaultSetpoints.heating.standby.setpoint	:= 2;
defaultSetpoints.heating.economy.setpoint	:= 3;
defaultSetpoints.cooling.comfort.setpoint	:= 2;
defaultSetpoints.cooling.standby.setpoint	:= 3;
defaultSetpoints.cooling.economy.setpoint	:= 4;
defaultSetpoints.co2.comfort.setpoint		:= 600;
defaultSetpoints.presenceDelayOff			:= 30;
defaultSetpoints.heating.pidSettings.KP		:= 1;
defaultSetpoints.heating.pidSettings.TN		:= 60;
defaultSetpoints.cooling.pidSettings.KP		:= 1;
defaultSetpoints.cooling.pidSettings.TN		:= 60;
defaultSetpoints.co2.pidSettings.KP			:= 20;
defaultSetpoints.co2.pidSettings.TN			:= 4000;
                            
                        
END_ACTION
END_PROGRAM

PROGRAM ClimateControl_547_2
  VAR
    climateController : FbMultiModeClimateControl_00_02;
    defaultSetpoints : typMultiModeClimateControllerDefaultSettings_00_01;
    dwConfigurationMask : DWORD := 2#0000_0000_0000_0000_0000_0001_0000_0010;
  END_VAR
  VAR_OUTPUT
    actualSetpointHeating : REAL;  (* Variabler kun for overvåking *)
    actualSetpointCooling : REAL;
    actualSetpointCo2 : REAL;
    meanTemp : REAL;
    meanCo2 : REAL;
    presence : BOOL;
    gainHeating : REAL;
    gainCooling : REAL;
    gainAirQuality : REAL;
    damperOutput : REAL;
    currentWorkingMode : enumMultiModeClimateActiveControlMode_00_01;
  END_VAR

                
    
// Innstillinger for rom:
IF (firstScan) THEN
    PersistentVars.typClimateControllerSettingsRoom547_2.ahuSystem		:= 001;
    PersistentVars.typClimateControllerSettingsRoom547_2.heatingSystem	:= 005;
    PersistentVars.typClimateControllerSettingsRoom547_2.coolingSystem	:= 005;
    defaultSetpoints 							:= PersistentVars.typClimateControlDefaultSettings;
    
// Hvis du ønsker egne innstillinger for rommet, kjør settings
    // settings();
END_IF

// Tilbakestill settpunkt (global kommando)
IF (GVL.initDefaultSettings) THEN
    climateController.setDefaultSetpoints();
END_IF

// Kjør funksjonsblokk
climateController(
    typController			:= typClimateControllerInterfaceRoom547_2, 
    typSettings				:= PersistentVars.typClimateControllerSettingsRoom547_2, 
    typDefaultSetpoints		:= defaultSetpoints,
    dwConfigurationMask		:= dwConfigurationMask            
);
        
// Registrer temperaturer
climateController.Temp          := PRG_KnxLine_2.M2_022_547_2_RMA6010_TMP_ACT.rValue_OUT;

// Registrer CO2
climateController.CO2          := PRG_KnxLine_2.M2_034_547_2_RMA6010_CO2_ACT.rValue_OUT;

// Registrer tilstedeværelse
climateController.Presence          := PRG_KnxLine_2.M2_010_547_2_RMA6010_MOV_ACT.xSwitch_OUT;

meanTemp					:= typClimateControllerInterfaceRoom547_2.actuators.heating.processValue;
meanCo2						:= climateController.Co2;
presence					:= climateController.Presence;

actualSetpointHeating 		:= typClimateControllerInterfaceRoom547_2.actuators.heating.setpoint;
gainHeating 				:= typClimateControllerInterfaceRoom547_2.actuators.heating.controlledVariable;

actualSetpointCooling 		:= typClimateControllerInterfaceRoom547_2.actuators.cooling.setpoint;
gainCooling 				:= typClimateControllerInterfaceRoom547_2.actuators.cooling.controlledVariable;

actualSetpointCo2			:= typClimateControllerInterfaceRoom547_2.actuators.airQuality.setpoint;
gainAirQuality				:= typClimateControllerInterfaceRoom547_2.actuators.airQuality.controlledVariable; 
damperOutput				:= typClimateControllerInterfaceRoom547_2.actuators.damper.setpoint;

currentWorkingMode			:= typClimateControllerInterfaceRoom547_2.currentMode;                   
                
                
              

ACTION settings:
                            
                                
defaultSetpoints.heating.comfort.setpoint	:= 21;
defaultSetpoints.heating.standby.setpoint	:= 2;
defaultSetpoints.heating.economy.setpoint	:= 3;
defaultSetpoints.cooling.comfort.setpoint	:= 2;
defaultSetpoints.cooling.standby.setpoint	:= 3;
defaultSetpoints.cooling.economy.setpoint	:= 4;
defaultSetpoints.co2.comfort.setpoint		:= 600;
defaultSetpoints.presenceDelayOff			:= 30;
defaultSetpoints.heating.pidSettings.KP		:= 1;
defaultSetpoints.heating.pidSettings.TN		:= 60;
defaultSetpoints.cooling.pidSettings.KP		:= 1;
defaultSetpoints.cooling.pidSettings.TN		:= 60;
defaultSetpoints.co2.pidSettings.KP			:= 20;
defaultSetpoints.co2.pidSettings.TN			:= 4000;
                            
                        
END_ACTION
END_PROGRAM

PROGRAM ClimateControl_544
  VAR
    climateController : FbMultiModeClimateControl_00_02;
    defaultSetpoints : typMultiModeClimateControllerDefaultSettings_00_01;
    dwConfigurationMask : DWORD := 2#0000_0000_0000_0000_0000_0001_0000_0010;
  END_VAR
  VAR_OUTPUT
    actualSetpointHeating : REAL;  (* Variabler kun for overvåking *)
    actualSetpointCooling : REAL;
    actualSetpointCo2 : REAL;
    meanTemp : REAL;
    meanCo2 : REAL;
    presence : BOOL;
    gainHeating : REAL;
    gainCooling : REAL;
    gainAirQuality : REAL;
    damperOutput : REAL;
    currentWorkingMode : enumMultiModeClimateActiveControlMode_00_01;
  END_VAR

                
    
// Innstillinger for rom:
IF (firstScan) THEN
    PersistentVars.typClimateControllerSettingsRoom544.ahuSystem		:= 001;
    PersistentVars.typClimateControllerSettingsRoom544.heatingSystem	:= 005;
    PersistentVars.typClimateControllerSettingsRoom544.coolingSystem	:= 005;
    defaultSetpoints 							:= PersistentVars.typClimateControlDefaultSettings;
    
// Hvis du ønsker egne innstillinger for rommet, kjør settings
    // settings();
END_IF

// Tilbakestill settpunkt (global kommando)
IF (GVL.initDefaultSettings) THEN
    climateController.setDefaultSetpoints();
END_IF

// Kjør funksjonsblokk
climateController(
    typController			:= typClimateControllerInterfaceRoom544, 
    typSettings				:= PersistentVars.typClimateControllerSettingsRoom544, 
    typDefaultSetpoints		:= defaultSetpoints,
    dwConfigurationMask		:= dwConfigurationMask            
);
        
// Registrer temperaturer
climateController.Temp          := PRG_KnxLine_2.M2_023_544_RMA6011_TMP_ACT.rValue_OUT;
climateController.Temp          := PRG_KnxLine_2.M2_024_544_RMA6012_TMP_ACT.rValue_OUT;

// Registrer CO2
climateController.CO2          := PRG_KnxLine_2.M2_035_544_RMA6011_CO2_ACT.rValue_OUT;
climateController.CO2          := PRG_KnxLine_2.M2_036_544_RMA6012_CO2_ACT.rValue_OUT;

// Registrer tilstedeværelse
climateController.Presence          := PRG_KnxLine_2.M2_011_544_RMA6011_MOV_ACT.xSwitch_OUT;
climateController.Presence          := PRG_KnxLine_2.M2_012_544_RMA6012_MOV_ACT.xSwitch_OUT;

meanTemp					:= typClimateControllerInterfaceRoom544.actuators.heating.processValue;
meanCo2						:= climateController.Co2;
presence					:= climateController.Presence;

actualSetpointHeating 		:= typClimateControllerInterfaceRoom544.actuators.heating.setpoint;
gainHeating 				:= typClimateControllerInterfaceRoom544.actuators.heating.controlledVariable;

actualSetpointCooling 		:= typClimateControllerInterfaceRoom544.actuators.cooling.setpoint;
gainCooling 				:= typClimateControllerInterfaceRoom544.actuators.cooling.controlledVariable;

actualSetpointCo2			:= typClimateControllerInterfaceRoom544.actuators.airQuality.setpoint;
gainAirQuality				:= typClimateControllerInterfaceRoom544.actuators.airQuality.controlledVariable; 
damperOutput				:= typClimateControllerInterfaceRoom544.actuators.damper.setpoint;

currentWorkingMode			:= typClimateControllerInterfaceRoom544.currentMode;                   
                
                
              

ACTION settings:
                            
                                
defaultSetpoints.heating.comfort.setpoint	:= 21;
defaultSetpoints.heating.standby.setpoint	:= 2;
defaultSetpoints.heating.economy.setpoint	:= 3;
defaultSetpoints.cooling.comfort.setpoint	:= 2;
defaultSetpoints.cooling.standby.setpoint	:= 3;
defaultSetpoints.cooling.economy.setpoint	:= 4;
defaultSetpoints.co2.comfort.setpoint		:= 600;
defaultSetpoints.presenceDelayOff			:= 30;
defaultSetpoints.heating.pidSettings.KP		:= 1;
defaultSetpoints.heating.pidSettings.TN		:= 60;
defaultSetpoints.cooling.pidSettings.KP		:= 1;
defaultSetpoints.cooling.pidSettings.TN		:= 60;
defaultSetpoints.co2.pidSettings.KP			:= 20;
defaultSetpoints.co2.pidSettings.TN			:= 4000;
                            
                        
END_ACTION
END_PROGRAM

PROGRAM PRG_ClimateControl

                
    ClimateControl_401();
ClimateControl_406();
ClimateControl_407();
ClimateControl_408();
ClimateControl_409();
ClimateControl_464();
ClimateControl_415();
ClimateControl_422();
ClimateControl_426_1();
ClimateControl_426_2();
ClimateControl_426_3();
ClimateControl_528();
ClimateControl_523();
ClimateControl_531();
ClimateControl_535_1();
ClimateControl_535_2();
ClimateControl_535_3();
ClimateControl_536();
ClimateControl_543();
ClimateControl_547_1();
ClimateControl_547_2();
ClimateControl_544();

                
              
END_PROGRAM

